C05449=1136.949,196.635,-63.220,-178.213,7.501,148.900
C05450=1136.954,196.386,-63.196,-178.216,7.499,148.901
C05451=1136.958,196.137,-63.172,-178.219,7.496,148.901
C05452=1136.963,195.889,-63.148,-178.222,7.493,148.901
C05453=1136.968,195.639,-63.124,-178.225,7.491,148.901
C05454=1136.973,195.391,-63.100,-178.227,7.488,148.901
C05455=1136.976,195.142,-63.076,-178.230,7.486,148.902
C05456=1136.981,194.893,-63.053,-178.233,7.483,148.902
C05457=1136.986,194.644,-63.028,-178.236,7.481,148.902
C05458=1136.990,194.396,-63.004,-178.239,7.478,148.902
C05459=1136.995,194.147,-62.980,-178.242,7.476,148.902
C05460=1137.000,193.898,-62.956,-178.244,7.474,148.903
C05461=1137.004,193.649,-62.933,-178.247,7.471,148.903
C05462=1137.009,193.401,-62.909,-178.250,7.468,148.903
C05463=1137.013,193.151,-62.885,-178.252,7.466,148.903
C05464=1137.017,192.903,-62.861,-178.256,7.464,148.904
C05465=1137.022,192.654,-62.838,-178.258,7.462,148.904
C05466=1137.026,192.405,-62.814,-178.261,7.459,148.904
C05467=1137.032,192.156,-62.790,-178.264,7.456,148.904
C05468=1137.036,191.908,-62.766,-178.267,7.454,148.905
C05469=1137.041,191.658,-62.742,-178.270,7.452,148.905
C05470=1137.045,191.410,-62.718,-178.273,7.449,148.905
C05471=1137.050,191.161,-62.695,-178.275,7.447,148.905
C05472=1137.055,190.912,-62.671,-178.278,7.444,148.905
C05473=1137.059,190.664,-62.647,-178.281,7.442,148.906
C05474=1137.064,190.415,-62.624,-178.284,7.440,148.906
C05475=1137.068,190.166,-62.600,-178.287,7.437,148.906
C05476=1137.073,189.917,-62.577,-178.290,7.434,148.906
C05477=1137.078,189.668,-62.553,-178.292,7.432,148.907
C05478=1137.082,189.420,-62.529,-178.295,7.429,148.907
C05479=1137.087,189.171,-62.506,-178.298,7.428,148.907
C05480=1137.091,188.922,-62.482,-178.301,7.425,148.907
C05481=1137.096,188.673,-62.459,-178.304,7.422,148.907
C05482=1137.101,188.424,-62.435,-178.306,7.420,148.908
C05483=1137.105,188.175,-62.412,-178.309,7.418,148.908
C05484=1137.110,187.926,-62.388,-178.312,7.416,148.908
C05485=1137.115,187.677,-62.365,-178.315,7.413,148.908
C05486=1137.119,187.429,-62.341,-178.318,7.410,148.909
C05487=1137.124,187.180,-62.318,-178.320,7.408,148.909
C05488=1137.128,186.931,-62.294,-178.323,7.405,148.909
C05489=1137.133,186.682,-62.271,-178.327,7.403,148.909
C05490=1137.137,186.433,-62.247,-178.329,7.401,148.909
C05491=1137.141,186.184,-62.224,-178.332,7.398,148.910
C05492=1137.146,185.935,-62.201,-178.334,7.396,148.910
C05493=1137.151,185.686,-62.177,-178.338,7.394,148.910
C05494=1137.156,185.437,-62.154,-178.341,7.391,148.911
C05495=1137.160,185.188,-62.131,-178.343,7.389,148.911
C05496=1137.165,184.939,-62.107,-178.346,7.387,148.911
C05497=1137.169,184.691,-62.084,-178.349,7.384,148.911
C05498=1137.173,184.442,-62.060,-178.352,7.382,148.912
C05499=1137.178,184.193,-62.037,-178.354,7.380,148.912
C05500=1137.183,183.944,-62.014,-178.357,7.377,148.912
C05501=1137.188,183.674,-61.989,-178.360,7.374,148.912
C05502=1137.193,183.405,-61.964,-178.363,7.372,148.913
C05503=1137.198,183.135,-61.939,-178.367,7.369,148.913
C05504=1137.203,182.866,-61.913,-178.370,7.366,148.913
C05505=1137.208,182.617,-61.890,-178.372,7.365,148.913
C05506=1137.212,182.368,-61.867,-178.375,7.362,148.914
C05507=1137.216,182.119,-61.844,-178.378,7.360,148.914
C05508=1137.221,181.869,-61.821,-178.381,7.358,148.914
C05509=1137.226,181.620,-61.798,-178.383,7.356,148.914
C05510=1137.231,181.372,-61.775,-178.387,7.353,148.915
C05511=1137.235,181.123,-61.752,-178.389,7.351,148.915
C05512=1137.240,180.874,-61.729,-178.392,7.348,148.915
C05513=1137.245,180.625,-61.705,-178.395,7.345,148.915
C05514=1137.249,180.377,-61.683,-178.398,7.344,148.916
C05515=1137.253,180.128,-61.659,-178.401,7.341,148.916
C05516=1137.259,179.879,-61.636,-178.403,7.339,148.916
C05517=1137.263,179.630,-61.614,-178.406,7.337,148.917
C05518=1137.268,179.381,-61.591,-178.409,7.335,148.917
C05519=1137.272,179.132,-61.568,-178.412,7.332,148.917
C05520=1137.276,178.883,-61.545,-178.414,7.330,148.917
C05521=1137.281,178.634,-61.521,-178.418,7.327,148.918
C05522=1137.286,178.385,-61.500,-178.421,7.325,148.918
C05523=1137.291,178.136,-61.476,-178.423,7.323,148.918
C05524=1137.295,177.887,-61.453,-178.426,7.320,148.918
C05525=1137.299,177.639,-61.430,-178.429,7.318,148.918
C05526=1137.305,177.390,-61.408,-178.432,7.316,148.919
C05527=1137.309,177.141,-61.385,-178.435,7.314,148.919
C05528=1137.313,176.892,-61.362,-178.437,7.311,148.919
C05529=1137.318,176.643,-61.338,-178.440,7.309,148.920
C05530=1137.323,176.394,-61.317,-178.443,7.306,148.920
C05531=1137.328,176.145,-61.293,-178.446,7.305,148.920
C05532=1137.332,175.897,-61.271,-178.449,7.302,148.921
C05533=1137.337,175.647,-61.248,-178.451,7.300,148.921
C05534=1137.341,175.399,-61.226,-178.454,7.298,148.921
C05535=1137.346,175.149,-61.203,-178.457,7.295,148.921
C05536=1137.350,174.900,-61.180,-178.460,7.293,148.922
C05537=1137.355,174.651,-61.157,-178.463,7.291,148.922
C05538=1137.360,174.403,-61.135,-178.465,7.288,148.922
C05539=1137.365,174.154,-61.112,-178.468,7.287,148.922
C05540=1137.369,173.904,-61.090,-178.471,7.284,148.923
C05541=1137.374,173.656,-61.067,-178.474,7.282,148.923
C05542=1137.378,173.407,-61.045,-178.477,7.279,148.923
C05543=1137.383,173.158,-61.021,-178.479,7.277,148.923
C05544=1137.388,172.909,-61.000,-178.483,7.275,148.924
C05545=1137.393,172.660,-60.976,-178.485,7.273,148.924
C05546=1137.397,172.411,-60.954,-178.488,7.270,148.924
C05547=1137.401,172.163,-60.932,-178.491,7.269,148.925
C05548=1137.406,171.913,-60.909,-178.494,7.266,148.925
C05549=1137.410,171.664,-60.886,-178.496,7.264,148.925
C05550=1137.416,171.415,-60.864,-178.500,7.261,148.925
C05551=1137.420,171.167,-60.841,-178.502,7.260,148.926
C05552=1137.425,170.918,-60.820,-178.505,7.257,148.926
C05553=1137.430,170.668,-60.797,-178.508,7.255,148.926
C05554=1137.434,170.420,-60.774,-178.511,7.253,148.927
C05555=1137.439,170.171,-60.753,-178.513,7.251,148.927
C05556=1137.444,169.921,-60.730,-178.517,7.248,148.927
C05557=1137.448,169.673,-60.707,-178.519,7.246,148.928
C05558=1137.453,169.424,-60.686,-178.522,7.244,148.928
C05559=1137.458,169.174,-60.663,-178.525,7.242,148.928
C05560=1137.462,168.926,-60.641,-178.528,7.240,148.928
C05561=1137.466,168.677,-60.618,-178.530,7.237,148.929
C05562=1137.472,168.428,-60.596,-178.533,7.235,148.929
C05563=1137.476,168.179,-60.573,-178.536,7.233,148.929
C05564=1137.480,167.930,-60.551,-178.539,7.231,148.929
C05565=1137.486,167.681,-60.529,-178.542,7.228,148.930
C05566=1137.490,167.432,-60.507,-178.545,7.227,148.930
C05567=1137.495,167.183,-60.485,-178.547,7.224,148.930
C05568=1137.499,166.934,-60.463,-178.550,7.222,148.931
C05569=1137.505,166.685,-60.440,-178.553,7.220,148.931
C05570=1137.509,166.436,-60.418,-178.556,7.217,148.931
C05571=1137.514,166.187,-60.397,-178.558,7.216,148.932
C05572=1137.518,165.938,-60.375,-178.562,7.213,148.932
C05573=1137.524,165.689,-60.352,-178.564,7.211,148.932
C05574=1137.527,165.440,-60.330,-178.567,7.208,148.932
C05575=1137.532,165.192,-60.308,-178.570,7.207,148.933
C05576=1137.537,164.942,-60.286,-178.573,7.205,148.933
C05577=1137.542,164.694,-60.264,-178.576,7.202,148.933
C05578=1137.546,164.444,-60.242,-178.578,7.200,148.934
C05579=1137.551,164.195,-60.220,-178.582,7.198,148.934
C05580=1137.556,163.946,-60.198,-178.584,7.196,148.934
C05581=1137.561,163.697,-60.176,-178.587,7.193,148.935
C05582=1137.565,163.448,-60.154,-178.590,7.192,148.935
C05583=1137.570,163.199,-60.132,-178.592,7.190,148.935
C05584=1137.574,162.950,-60.110,-178.595,7.187,148.935
C05585=1137.579,162.702,-60.089,-178.598,7.185,148.936
C05586=1137.583,162.452,-60.067,-178.601,7.183,148.936
C05587=1137.588,162.204,-60.045,-178.604,7.181,148.936
C05588=1137.592,161.954,-60.023,-178.606,7.179,148.937
C05589=1137.598,161.705,-60.001,-178.610,7.176,148.937
C05590=1137.602,161.456,-59.978,-178.612,7.175,148.937
C05591=1137.607,161.207,-59.957,-178.615,7.172,148.938
C05592=1137.612,160.959,-59.935,-178.618,7.170,148.938
C05593=1137.616,160.709,-59.913,-178.620,7.168,148.938
C05594=1137.621,160.461,-59.891,-178.624,7.166,148.939
C05595=1137.625,160.211,-59.869,-178.626,7.164,148.939
C05596=1137.630,159.962,-59.848,-178.629,7.161,148.939
C05597=1137.635,159.713,-59.827,-178.632,7.160,148.940
C05598=1137.640,159.464,-59.805,-178.635,7.158,148.940
C05599=1137.644,159.215,-59.783,-178.638,7.155,148.940
C05600=1137.649,158.966,-59.761,-178.640,7.153,148.941
C05601=1137.654,158.717,-59.739,-178.644,7.151,148.941
C05602=1137.659,158.468,-59.718,-178.646,7.149,148.941
C05603=1137.663,158.219,-59.696,-178.649,7.147,148.941
C05604=1137.668,157.970,-59.675,-178.652,7.145,148.942
C05605=1137.673,157.701,-59.652,-178.655,7.143,148.942
C05606=1137.678,157.432,-59.628,-178.658,7.140,148.943
C05607=1137.683,157.163,-59.605,-178.661,7.138,148.943
C05608=1137.688,156.894,-59.582,-178.664,7.136,148.943
C05609=1137.693,156.645,-59.560,-178.667,7.134,148.944
C05610=1137.698,156.397,-59.538,-178.669,7.131,148.944
C05611=1137.702,156.147,-59.517,-178.672,7.130,148.944
C05612=1137.706,155.898,-59.496,-178.675,7.127,148.945
C05613=1137.711,155.650,-59.474,-178.678,7.126,148.945
C05614=1137.716,155.400,-59.453,-178.680,7.123,148.945
C05615=1137.721,155.151,-59.431,-178.684,7.121,148.945
C05616=1137.726,154.903,-59.409,-178.686,7.119,148.946
C05617=1137.730,154.653,-59.388,-178.689,7.118,148.946
C05618=1137.735,154.404,-59.366,-178.692,7.115,148.947
C05619=1137.740,154.155,-59.346,-178.695,7.113,148.947
C05620=1137.744,153.906,-59.324,-178.697,7.111,148.947
C05621=1137.749,153.656,-59.303,-178.701,7.109,148.947
C05622=1137.754,153.408,-59.281,-178.703,7.107,148.948
C05623=1137.759,153.159,-59.260,-178.706,7.105,148.948
C05624=1137.763,152.910,-59.239,-178.709,7.102,148.948
C05625=1137.767,152.661,-59.217,-178.712,7.101,148.949
C05626=1137.773,152.412,-59.196,-178.714,7.099,148.949
C05627=1137.777,152.163,-59.175,-178.718,7.096,148.950
C05628=1137.783,151.914,-59.154,-178.720,7.095,148.950
C05629=1137.786,151.665,-59.132,-178.723,7.093,148.950
C05630=1137.791,151.415,-59.111,-178.726,7.090,148.950
C05631=1137.796,151.166,-59.090,-178.729,7.088,148.951
C05632=1137.801,150.918,-59.069,-178.731,7.087,148.951
C05633=1137.806,150.669,-59.048,-178.735,7.084,148.952
C05634=1137.810,150.419,-59.026,-178.737,7.082,148.952
C05635=1137.815,150.170,-59.005,-178.740,7.080,148.952
C05636=1137.820,149.921,-58.985,-178.743,7.078,148.953
C05637=1137.825,149.672,-58.963,-178.746,7.076,148.953
C05638=1137.830,149.423,-58.942,-178.748,7.075,148.953
C05639=1137.834,149.173,-58.921,-178.751,7.073,148.954
C05640=1137.838,148.925,-58.900,-178.754,7.070,148.954
C05641=1137.844,148.676,-58.879,-178.757,7.068,148.954
C05642=1137.848,148.427,-58.858,-178.759,7.067,148.955
C05643=1137.853,148.178,-58.837,-178.763,7.064,148.955
C05644=1137.858,147.929,-58.816,-178.765,7.062,148.955
C05645=1137.862,147.679,-58.795,-178.768,7.061,148.956
C05646=1137.867,147.430,-58.773,-178.770,7.059,148.956
C05647=1137.871,147.181,-58.753,-178.774,7.056,148.956
C05648=1137.876,146.932,-58.732,-178.776,7.054,148.957
C05649=1137.882,146.683,-58.711,-178.779,7.053,148.957
C05650=1137.886,146.434,-58.691,-178.782,7.050,148.957
C05651=1137.891,146.185,-58.669,-178.785,7.048,148.958
C05652=1137.895,145.936,-58.649,-178.788,7.047,148.958
C05653=1137.900,145.687,-58.628,-178.790,7.045,148.958
C05654=1137.904,145.437,-58.607,-178.793,7.042,148.959
C05655=1137.910,145.188,-58.586,-178.796,7.040,148.959
C05656=1137.914,144.940,-58.564,-178.799,7.039,148.959
C05657=1137.919,144.691,-58.544,-178.802,7.036,148.960
C05658=1137.924,144.441,-58.523,-178.805,7.035,148.960
C05659=1137.928,144.192,-58.503,-178.807,7.033,148.961
C05660=1137.934,143.943,-58.482,-178.810,7.031,148.961
C05661=1137.938,143.694,-58.461,-178.813,7.028,148.961
C05662=1137.943,143.445,-58.440,-178.816,7.027,148.962
C05663=1137.948,143.196,-58.420,-178.818,7.025,148.962
C05664=1137.952,142.947,-58.399,-178.821,7.023,148.962
C05665=1137.957,142.698,-58.378,-178.824,7.021,148.963
C05666=1137.962,142.449,-58.358,-178.827,7.019,148.963
C05667=1137.967,142.200,-58.337,-178.830,7.017,148.963
C05668=1137.971,141.951,-58.317,-178.832,7.015,148.964
C05669=1137.976,141.701,-58.296,-178.835,7.013,148.964
C05670=1137.980,141.452,-58.275,-178.838,7.011,148.964
C05671=1137.985,141.203,-58.255,-178.841,7.009,148.965
C05672=1137.990,140.953,-58.234,-178.844,7.008,148.965
C05673=1137.994,140.705,-58.213,-178.846,7.006,148.966
C05674=1138.000,140.455,-58.192,-178.850,7.003,148.966
C05675=1138.004,140.206,-58.172,-178.852,7.002,148.966
C05676=1138.008,139.957,-58.152,-178.855,7.000,148.967
C05677=1138.014,139.708,-58.131,-178.857,6.998,148.967
C05678=1138.019,139.460,-58.111,-178.861,6.995,148.967
C05679=1138.023,139.211,-58.090,-178.863,6.994,148.968
C05680=1138.028,138.962,-58.069,-178.866,6.992,148.968
C05681=1138.033,138.712,-58.050,-178.869,6.990,148.968
C05682=1138.037,138.463,-58.029,-178.871,6.989,148.969
C05683=1138.043,138.214,-58.008,-178.875,6.986,148.969
C05684=1138.047,137.965,-57.988,-178.878,6.984,148.970
C05685=1138.051,137.716,-57.968,-178.880,6.983,148.970
C05686=1138.057,137.466,-57.947,-178.883,6.981,148.970
C05687=1138.061,137.217,-57.927,-178.886,6.978,148.971
C05688=1138.066,136.968,-57.907,-178.889,6.976,148.971
C05689=1138.070,136.719,-57.886,-178.891,6.975,148.971
C05690=1138.075,136.470,-57.865,-178.894,6.973,148.972
C05691=1138.080,136.220,-57.846,-178.897,6.971,148.972
C05692=1138.085,135.972,-57.825,-178.900,6.969,148.973
C05693=1138.089,135.723,-57.805,-178.903,6.967,148.973
C05694=1138.095,135.473,-57.785,-178.905,6.965,148.973
C05695=1138.100,135.224,-57.765,-178.908,6.964,148.974
C05696=1138.104,134.975,-57.744,-178.911,6.962,148.974
C05697=1138.109,134.726,-57.725,-178.914,6.960,148.975
C05698=1138.114,134.477,-57.704,-178.917,6.958,148.975
C05699=1138.118,134.228,-57.683,-178.920,6.956,148.975
C05700=1138.123,133.978,-57.664,-178.922,6.954,148.976
C05701=1138.128,133.729,-57.643,-178.925,6.953,148.976
C05702=1138.133,133.481,-57.623,-178.928,6.951,148.976
C05703=1138.137,133.231,-57.604,-178.931,6.948,148.977
C05704=1138.142,132.982,-57.583,-178.933,6.946,148.977
C05705=1138.147,132.733,-57.563,-178.936,6.945,148.977
C05706=1138.152,132.484,-57.543,-178.939,6.943,148.978
C05707=1138.156,132.234,-57.523,-178.942,6.941,148.978
C05708=1138.161,131.986,-57.503,-178.944,6.940,148.979
C05709=1138.167,131.717,-57.481,-178.948,6.937,148.979
C05710=1138.172,131.449,-57.459,-178.950,6.936,148.979
C05711=1138.177,131.180,-57.438,-178.954,6.933,148.980
C05712=1138.182,130.911,-57.417,-178.957,6.932,148.980
C05713=1138.187,130.662,-57.396,-178.960,6.930,148.981
C05714=1138.191,130.413,-57.377,-178.962,6.928,148.981
C05715=1138.196,130.164,-57.356,-178.965,6.927,148.982
C05716=1138.201,129.915,-57.337,-178.968,6.924,148.982
C05717=1138.206,129.666,-57.317,-178.971,6.922,148.982
C05718=1138.210,129.416,-57.297,-178.973,6.920,148.983
C05719=1138.215,129.167,-57.277,-178.976,6.919,148.983
C05720=1138.220,128.919,-57.257,-178.979,6.917,148.983
C05721=1138.225,128.669,-57.238,-178.981,6.915,148.984
C05722=1138.229,128.420,-57.217,-178.984,6.914,148.984
C05723=1138.234,128.170,-57.198,-178.987,6.911,148.985
C05724=1138.239,127.922,-57.178,-178.990,6.909,148.985
C05725=1138.244,127.673,-57.158,-178.993,6.908,148.985
C05726=1138.249,127.423,-57.138,-178.996,6.906,148.986
C05727=1138.253,127.173,-57.119,-178.998,6.904,148.986
C05728=1138.258,126.925,-57.099,-179.001,6.903,148.986
C05729=1138.263,126.676,-57.079,-179.004,6.901,148.987
C05730=1138.268,126.426,-57.059,-179.007,6.899,148.987
C05731=1138.273,126.177,-57.040,-179.010,6.897,148.988
C05732=1138.278,125.928,-57.020,-179.013,6.895,148.988
C05733=1138.282,125.679,-57.000,-179.015,6.893,148.988
C05734=1138.287,125.429,-56.980,-179.018,6.892,148.989
C05735=1138.293,125.180,-56.961,-179.021,6.890,148.989
C05736=1138.297,124.931,-56.941,-179.023,6.888,148.990
C05737=1138.302,124.682,-56.921,-179.026,6.887,148.990
C05738=1138.306,124.433,-56.902,-179.029,6.885,148.990
C05739=1138.311,124.184,-56.883,-179.032,6.883,148.991
C05740=1138.316,123.934,-56.863,-179.035,6.881,148.991
C05741=1138.321,123.686,-56.843,-179.038,6.879,148.992
C05742=1138.326,123.436,-56.823,-179.040,6.877,148.992
C05743=1138.330,123.187,-56.804,-179.043,6.876,148.992
C05744=1138.336,122.938,-56.784,-179.046,6.874,148.993
C05745=1138.340,122.689,-56.765,-179.049,6.872,148.993
C05746=1138.344,122.439,-56.746,-179.051,6.871,148.994
C05747=1138.350,122.190,-56.726,-179.054,6.869,148.994
C05748=1138.355,121.941,-56.707,-179.057,6.867,148.994
C05749=1138.359,121.691,-56.687,-179.059,6.866,148.995
C05750=1138.364,121.442,-56.668,-179.062,6.864,148.995
C05751=1138.369,121.193,-56.649,-179.066,6.861,148.996
C05752=1138.374,120.945,-56.629,-179.068,6.860,148.996
C05753=1138.378,120.695,-56.609,-179.071,6.858,148.996
C05754=1138.383,120.445,-56.589,-179.074,6.856,148.997
C05755=1138.388,120.197,-56.571,-179.076,6.855,148.997
C05756=1138.392,119.947,-56.551,-179.079,6.853,148.998
C05757=1138.398,119.698,-56.532,-179.082,6.851,148.998
C05758=1138.403,119.448,-56.513,-179.085,6.850,148.998
C05759=1138.407,119.200,-56.494,-179.088,6.848,148.999
C05760=1138.412,118.950,-56.474,-179.091,6.847,149.000
C05761=1138.417,118.701,-56.455,-179.093,6.845,149.000
C05762=1138.422,118.452,-56.436,-179.096,6.843,149.000
C05763=1138.426,118.202,-56.416,-179.099,6.841,149.001
C05764=1138.432,117.954,-56.397,-179.101,6.840,149.001
C05765=1138.436,117.704,-56.378,-179.104,6.838,149.002
C05766=1138.441,117.455,-56.359,-179.107,6.836,149.002
C05767=1138.446,117.206,-56.339,-179.110,6.834,149.002
C05768=1138.450,116.957,-56.320,-179.113,6.832,149.003
C05769=1138.455,116.707,-56.302,-179.116,6.831,149.003
C05770=1138.461,116.458,-56.282,-179.118,6.829,149.004
C05771=1138.465,116.209,-56.263,-179.121,6.827,149.004
C05772=1138.470,115.960,-56.244,-179.124,6.825,149.004
C05773=1138.475,115.711,-56.224,-179.127,6.824,149.005
C05774=1138.480,115.461,-56.206,-179.129,6.822,149.005
C05775=1138.484,115.212,-56.187,-179.132,6.820,149.006
C05776=1138.489,114.963,-56.168,-179.135,6.819,149.006
C05777=1138.494,114.714,-56.148,-179.138,6.817,149.006
C05778=1138.499,114.464,-56.130,-179.140,6.815,149.007
C05779=1138.503,114.215,-56.111,-179.143,6.814,149.007
C05780=1138.509,113.966,-56.091,-179.146,6.812,149.008
C05781=1138.513,113.717,-56.072,-179.149,6.811,149.008
C05782=1138.518,113.467,-56.054,-179.152,6.809,149.009
C05783=1138.523,113.219,-56.035,-179.154,6.807,149.009
C05784=1138.528,112.969,-56.015,-179.157,6.806,149.009
C05785=1138.533,112.720,-55.997,-179.160,6.804,149.010
C05786=1138.538,112.471,-55.978,-179.163,6.802,149.010
C05787=1138.543,112.222,-55.958,-179.165,6.801,149.011
C05788=1138.547,111.972,-55.940,-179.168,6.799,149.011
C05789=1138.552,111.723,-55.921,-179.171,6.797,149.012
C05790=1138.557,111.474,-55.903,-179.173,6.796,149.012
C05791=1138.562,111.224,-55.883,-179.176,6.794,149.012
C05792=1138.567,110.976,-55.864,-179.179,6.792,149.013
C05793=1138.572,110.725,-55.845,-179.182,6.791,149.013
C05794=1138.576,110.477,-55.827,-179.185,6.789,149.014
C05795=1138.582,110.227,-55.808,-179.188,6.787,149.014
C05796=1138.586,109.978,-55.789,-179.190,6.786,149.015
C05797=1138.591,109.729,-55.771,-179.193,6.784,149.015
C05798=1138.596,109.479,-55.752,-179.196,6.782,149.015
C05799=1138.601,109.230,-55.734,-179.199,6.781,149.016
C05800=1138.606,108.981,-55.714,-179.201,6.779,149.016
C05801=1138.610,108.731,-55.696,-179.204,6.777,149.017
C05802=1138.615,108.483,-55.677,-179.207,6.776,149.017
C05803=1138.621,108.233,-55.659,-179.209,6.774,149.017
C05804=1138.625,107.984,-55.640,-179.212,6.772,149.018
C05805=1138.630,107.735,-55.621,-179.215,6.771,149.019
C05806=1138.635,107.486,-55.602,-179.218,6.769,149.019
C05807=1138.639,107.236,-55.584,-179.221,6.768,149.019
C05808=1138.644,106.987,-55.565,-179.224,6.766,149.020
C05809=1138.649,106.738,-55.547,-179.226,6.764,149.020
C05810=1138.654,106.488,-55.528,-179.229,6.763,149.021
C05811=1138.659,106.239,-55.509,-179.232,6.761,149.021
C05812=1138.664,105.990,-55.491,-179.235,6.759,149.021
C05813=1138.668,105.721,-55.471,-179.238,6.758,149.022
C05814=1138.674,105.453,-55.451,-179.240,6.756,149.022
C05815=1138.679,105.185,-55.431,-179.243,6.755,149.023
C05816=1138.685,104.917,-55.411,-179.246,6.753,149.023
C05817=1138.690,104.667,-55.393,-179.249,6.752,149.024
C05818=1138.694,104.418,-55.374,-179.252,6.750,149.024
C05819=1138.699,104.169,-55.356,-179.255,6.748,149.025
C05820=1138.704,103.919,-55.338,-179.257,6.747,149.025
C05821=1138.708,103.670,-55.318,-179.260,6.745,149.026
C05822=1138.713,103.421,-55.301,-179.263,6.743,149.026
C05823=1138.719,103.172,-55.282,-179.266,6.742,149.026
C05824=1138.724,102.922,-55.264,-179.268,6.740,149.027
C05825=1138.728,102.673,-55.245,-179.271,6.738,149.027
C05826=1138.733,102.424,-55.227,-179.274,6.737,149.028
C05827=1138.738,102.174,-55.208,-179.277,6.735,149.028
C05828=1138.743,101.925,-55.190,-179.280,6.734,149.029
C05829=1138.748,101.676,-55.172,-179.282,6.732,149.029
C05830=1138.753,101.426,-55.154,-179.285,6.730,149.029
C05831=1138.757,101.178,-55.135,-179.287,6.729,149.030
C05832=1138.763,100.928,-55.117,-179.290,6.728,149.030
C05833=1138.768,100.679,-55.099,-179.293,6.726,149.031
C05834=1138.773,100.430,-55.081,-179.296,6.725,149.031
C05835=1138.777,100.180,-55.062,-179.299,6.723,149.032
C05836=1138.782,99.931,-55.044,-179.302,6.721,149.032
C05837=1138.787,99.682,-55.026,-179.304,6.720,149.033
C05838=1138.792,99.432,-55.009,-179.307,6.718,149.033
C05839=1138.797,99.184,-54.989,-179.310,6.716,149.033
C05840=1138.801,98.934,-54.971,-179.313,6.715,149.034
C05841=1138.806,98.684,-54.953,-179.316,6.713,149.035
C05842=1138.811,98.435,-54.935,-179.318,6.712,149.035
C05843=1138.816,98.186,-54.917,-179.321,6.711,149.035
C05844=1138.821,97.937,-54.899,-179.323,6.709,149.036
C05845=1138.826,97.688,-54.881,-179.326,6.707,149.036
C05846=1138.831,97.439,-54.863,-179.329,6.706,149.037
C05847=1138.835,97.189,-54.845,-179.332,6.704,149.037
C05848=1138.840,96.940,-54.827,-179.335,6.703,149.038
C05849=1138.845,96.690,-54.809,-179.337,6.701,149.038
C05850=1138.850,96.441,-54.791,-179.340,6.699,149.038
C05851=1138.855,96.192,-54.773,-179.343,6.698,149.039
C05852=1138.860,95.942,-54.755,-179.345,6.697,149.039
C05853=1138.865,95.693,-54.737,-179.348,6.696,149.040
C05854=1138.870,95.444,-54.719,-179.351,6.694,149.040
C05855=1138.875,95.194,-54.701,-179.354,6.692,149.041
C05856=1138.880,94.945,-54.683,-179.356,6.691,149.041
C05857=1138.884,94.696,-54.665,-179.359,6.689,149.042
C05858=1138.889,94.446,-54.647,-179.362,6.687,149.042
C05859=1138.894,94.197,-54.629,-179.365,6.686,149.042
C05860=1138.899,93.948,-54.611,-179.367,6.685,149.043
C05861=1138.904,93.698,-54.594,-179.370,6.683,149.044
C05862=1138.909,93.449,-54.576,-179.373,6.682,149.044
C05863=1138.914,93.200,-54.558,-179.376,6.680,149.044
C05864=1138.919,92.951,-54.540,-179.378,6.678,149.045
C05865=1138.923,92.702,-54.522,-179.381,6.677,149.045
C05866=1138.929,92.452,-54.505,-179.384,6.675,149.046
C05867=1138.934,92.203,-54.487,-179.386,6.675,149.046
C05868=1138.939,91.953,-54.469,-179.389,6.673,149.047
C05869=1138.943,91.704,-54.451,-179.392,6.671,149.047
C05870=1138.949,91.455,-54.434,-179.395,6.670,149.048
C05871=1138.954,91.205,-54.416,-179.398,6.668,149.048
C05872=1138.958,90.956,-54.398,-179.401,6.667,149.049
C05873=1138.963,90.707,-54.380,-179.403,6.666,149.049
C05874=1138.968,90.458,-54.363,-179.405,6.664,149.049
C05875=1138.973,90.208,-54.345,-179.408,6.662,149.050
C05876=1138.978,89.959,-54.327,-179.411,6.661,149.051
C05877=1138.983,89.709,-54.310,-179.414,6.659,149.051
C05878=1138.988,89.460,-54.292,-179.417,6.658,149.051
C05879=1138.992,89.211,-54.274,-179.420,6.656,149.052
C05880=1138.997,88.962,-54.257,-179.422,6.655,149.052
C05881=1139.002,88.712,-54.239,-179.425,6.654,149.053
C05882=1139.007,88.463,-54.222,-179.428,6.652,149.053
C05883=1139.012,88.213,-54.204,-179.430,6.651,149.054
C05884=1139.016,87.965,-54.187,-179.433,6.649,149.054
C05885=1139.022,87.715,-54.169,-179.435,6.648,149.055
C05886=1139.027,87.466,-54.151,-179.438,6.646,149.055
C05887=1139.032,87.216,-54.134,-179.441,6.645,149.056
C05888=1139.037,86.967,-54.116,-179.444,6.643,149.056
C05889=1139.041,86.717,-54.099,-179.447,6.642,149.056
C05890=1139.046,86.468,-54.081,-179.450,6.640,149.057
C05891=1139.051,86.219,-54.063,-179.452,6.639,149.057
C05892=1139.056,85.969,-54.046,-179.455,6.638,149.058
C05893=1139.060,85.720,-54.029,-179.458,6.636,149.058
C05894=1139.066,85.470,-54.012,-179.460,6.635,149.059
C05895=1139.071,85.221,-53.994,-179.463,6.633,149.059
C05896=1139.076,84.972,-53.977,-179.465,6.632,149.060
C05897=1139.081,84.723,-53.960,-179.469,6.631,149.060
C05898=1139.086,84.473,-53.942,-179.471,6.629,149.061
C05899=1139.090,84.224,-53.925,-179.474,6.628,149.061
C05900=1139.095,83.975,-53.907,-179.477,6.626,149.062
C05901=1139.100,83.725,-53.890,-179.479,6.625,149.062
C05902=1139.105,83.476,-53.873,-179.482,6.624,149.063
C05903=1139.110,83.226,-53.855,-179.485,6.622,149.063
C05904=1139.116,82.977,-53.839,-179.488,6.620,149.064
C05905=1139.120,82.728,-53.821,-179.490,6.620,149.064
C05906=1139.125,82.478,-53.804,-179.493,6.618,149.065
C05907=1139.130,82.229,-53.787,-179.496,6.617,149.065
C05908=1139.134,81.980,-53.769,-179.498,6.615,149.065
C05909=1139.140,81.730,-53.752,-179.501,6.613,149.066
C05910=1139.144,81.481,-53.735,-179.503,6.612,149.066
C05911=1139.150,81.232,-53.718,-179.507,6.611,149.067
C05912=1139.155,80.982,-53.700,-179.509,6.609,149.067
C05913=1139.159,80.733,-53.684,-179.512,6.608,149.068
C05914=1139.164,80.484,-53.666,-179.514,6.607,149.068
C05915=1139.169,80.234,-53.649,-179.517,6.606,149.069
C05916=1139.174,79.985,-53.632,-179.520,6.604,149.069
C05917=1139.180,79.716,-53.614,-179.523,6.602,149.070
C05918=1139.185,79.448,-53.595,-179.526,6.601,149.070
C05919=1139.190,79.179,-53.577,-179.529,6.599,149.071
C05920=1139.195,78.911,-53.559,-179.532,6.598,149.071
C05921=1139.200,78.662,-53.541,-179.535,6.596,149.072
C05922=1139.205,78.413,-53.525,-179.537,6.596,149.072
C05923=1139.210,78.163,-53.507,-179.540,6.594,149.073
C05924=1139.216,77.913,-53.490,-179.542,6.592,149.073
C05925=1139.220,77.664,-53.474,-179.546,6.591,149.074
C05926=1139.224,77.415,-53.456,-179.548,6.590,149.074
C05927=1139.230,77.166,-53.439,-179.551,6.588,149.075
C05928=1139.235,76.916,-53.423,-179.553,6.587,149.075
C05929=1139.240,76.667,-53.405,-179.557,6.585,149.076
C05930=1139.245,76.418,-53.389,-179.559,6.585,149.076
C05931=1139.250,76.168,-53.372,-179.561,6.583,149.077
C05932=1139.255,75.919,-53.355,-179.564,6.581,149.077
C05933=1139.260,75.669,-53.338,-179.567,6.581,149.078
C05934=1139.265,75.420,-53.321,-179.570,6.579,149.078
C05935=1139.270,75.170,-53.304,-179.572,6.578,149.079
C05936=1139.274,74.921,-53.287,-179.575,6.576,149.079
C05937=1139.279,74.672,-53.270,-179.578,6.575,149.080
C05938=1139.285,74.423,-53.253,-179.580,6.574,149.080
C05939=1139.289,74.173,-53.237,-179.583,6.572,149.081
C05940=1139.294,73.923,-53.219,-179.586,6.570,149.081
C05941=1139.299,73.675,-53.203,-179.589,6.570,149.082
C05942=1139.304,73.425,-53.186,-179.591,6.568,149.082
C05943=1139.309,73.175,-53.169,-179.594,6.567,149.083
C05944=1139.314,72.927,-53.153,-179.596,6.566,149.083
C05945=1139.319,72.676,-53.137,-179.599,6.564,149.084
C05946=1139.324,72.427,-53.120,-179.602,6.563,149.084
C05947=1139.329,72.178,-53.103,-179.604,6.562,149.084
C05948=1139.334,71.928,-53.087,-179.607,6.560,149.085
C05949=1139.339,71.679,-53.069,-179.610,6.559,149.086
C05950=1139.344,71.430,-53.053,-179.613,6.557,149.086
C05951=1139.348,71.180,-53.036,-179.615,6.557,149.086
C05952=1139.354,70.931,-53.019,-179.618,6.555,149.087
C05953=1139.359,70.682,-53.003,-179.621,6.554,149.088
C05954=1139.363,70.432,-52.986,-179.623,6.553,149.088
C05955=1139.369,70.182,-52.970,-179.626,6.551,149.088
C05956=1139.374,69.933,-52.953,-179.629,6.550,149.089
C05957=1139.378,69.684,-52.937,-179.632,6.549,149.089
C05958=1139.383,69.435,-52.920,-179.634,6.547,149.090
C05959=1139.389,69.185,-52.903,-179.637,6.546,149.090
C05960=1139.393,68.936,-52.886,-179.640,6.545,149.091
C05961=1139.398,68.686,-52.871,-179.642,6.544,149.091
C05962=1139.403,68.437,-52.854,-179.645,6.542,149.092
C05963=1139.409,68.188,-52.837,-179.647,6.541,149.092
C05964=1139.413,67.938,-52.821,-179.651,6.540,149.093
C05965=1139.418,67.688,-52.805,-179.653,6.538,149.093
C05966=1139.423,67.439,-52.788,-179.656,6.536,149.094
C05967=1139.428,67.190,-52.772,-179.658,6.536,149.094
C05968=1139.433,66.941,-52.755,-179.661,6.534,149.095
C05969=1139.438,66.691,-52.739,-179.664,6.533,149.095
C05970=1139.443,66.442,-52.722,-179.666,6.532,149.096
C05971=1139.448,66.192,-52.706,-179.670,6.531,149.096
C05972=1139.453,65.943,-52.690,-179.672,6.530,149.097
C05973=1139.458,65.693,-52.674,-179.674,6.528,149.097
C05974=1139.463,65.444,-52.656,-179.677,6.526,149.098
C05975=1139.468,65.194,-52.641,-179.680,6.526,149.098
C05976=1139.473,64.945,-52.624,-179.683,6.524,149.099
C05977=1139.478,64.696,-52.608,-179.685,6.523,149.099
C05978=1139.483,64.446,-52.592,-179.688,6.522,149.100
C05979=1139.488,64.197,-52.575,-179.691,6.520,149.100
C05980=1139.492,63.948,-52.559,-179.693,6.519,149.101
C05981=1139.498,63.698,-52.543,-179.696,6.518,149.101
C05982=1139.502,63.449,-52.527,-179.699,6.517,149.102
C05983=1139.508,63.199,-52.510,-179.702,6.515,149.102
C05984=1139.513,62.949,-52.494,-179.704,6.514,149.103
C05985=1139.518,62.700,-52.478,-179.707,6.513,149.103
C05986=1139.522,62.451,-52.461,-179.709,6.512,149.104
C05987=1139.528,62.202,-52.445,-179.712,6.510,149.104
C05988=1139.532,61.952,-52.429,-179.715,6.509,149.105
C05989=1139.537,61.703,-52.413,-179.717,6.508,149.105
C05990=1139.542,61.453,-52.397,-179.720,6.507,149.106
C05991=1139.547,61.204,-52.381,-179.723,6.505,149.106
C05992=1139.553,60.955,-52.365,-179.725,6.505,149.107
C05993=1139.557,60.705,-52.348,-179.728,6.503,149.107
C05994=1139.563,60.456,-52.333,-179.730,6.502,149.108
C05995=1139.567,60.206,-52.317,-179.734,6.501,149.109
C05996=1139.572,59.957,-52.301,-179.736,6.499,149.109
C05997=1139.577,59.707,-52.285,-179.738,6.498,149.109
C05998=1139.582,59.458,-52.268,-179.741,6.497,149.110
C05999=1139.587,59.208,-52.252,-179.744,6.495,149.111
C06000=1139.592,58.959,-52.236,-179.747,6.495,149.111
C06001=1139.598,58.710,-52.220,-179.749,6.493,149.111
C06002=1139.602,58.460,-52.204,-179.752,6.492,149.112
C06003=1139.607,58.211,-52.188,-179.755,6.491,149.112
C06004=1139.612,57.961,-52.172,-179.758,6.489,149.113
C06005=1139.618,57.711,-52.157,-179.760,6.489,149.114
C06006=1139.623,57.463,-52.140,-179.763,6.487,149.114
C06007=1139.627,57.212,-52.124,-179.765,6.486,149.114
C06008=1139.633,56.963,-52.109,-179.768,6.485,149.115
C06009=1139.637,56.714,-52.093,-179.771,6.483,149.116
C06010=1139.642,56.464,-52.077,-179.773,6.482,149.116
C06011=1139.647,56.215,-52.062,-179.776,6.481,149.116
C06012=1139.652,55.966,-52.045,-179.779,6.480,149.117
C06013=1139.657,55.716,-52.029,-179.781,6.479,149.118
C06014=1139.663,55.467,-52.014,-179.784,6.478,149.118
C06015=1139.667,55.217,-51.998,-179.787,6.477,149.119
C06016=1139.672,54.968,-51.981,-179.790,6.475,149.119
C06017=1139.678,54.718,-51.966,-179.792,6.474,149.120
C06018=1139.682,54.469,-51.950,-179.795,6.473,149.120
C06019=1139.687,54.219,-51.935,-179.797,6.472,149.121
C06020=1139.692,53.970,-51.919,-179.800,6.470,149.121
C06021=1139.698,53.701,-51.902,-179.803,6.469,149.122
C06022=1139.703,53.432,-51.885,-179.805,6.468,149.122
C06023=1139.709,53.164,-51.868,-179.808,6.467,149.123
C06024=1139.714,52.895,-51.851,-179.811,6.465,149.123
C06025=1139.719,52.646,-51.836,-179.814,6.464,149.124
C06026=1139.724,52.396,-51.820,-179.817,6.463,149.124
C06027=1139.729,52.147,-51.804,-179.819,6.462,149.125
C06028=1139.734,51.898,-51.788,-179.822,6.461,149.126
C06029=1139.740,51.648,-51.772,-179.825,6.459,149.126
C06030=1139.744,51.399,-51.757,-179.827,6.459,149.126
C06031=1139.749,51.149,-51.741,-179.830,6.457,149.127
C06032=1139.754,50.900,-51.726,-179.832,6.457,149.128
C06033=1139.759,50.650,-51.710,-179.835,6.455,149.128
C06034=1139.764,50.401,-51.695,-179.837,6.454,149.128
C06035=1139.769,50.151,-51.679,-179.840,6.453,149.129
C06036=1139.775,49.902,-51.664,-179.843,6.451,149.130
C06037=1139.779,49.652,-51.648,-179.845,6.450,149.130
C06038=1139.784,49.403,-51.633,-179.849,6.449,149.131
C06039=1139.789,49.153,-51.617,-179.851,6.448,149.131
C06040=1139.794,48.904,-51.602,-179.854,6.447,149.132
C06041=1139.799,48.654,-51.586,-179.856,6.446,149.132
C06042=1139.804,48.405,-51.571,-179.859,6.444,149.133
C06043=1139.810,48.155,-51.555,-179.861,6.444,149.133
C06044=1139.814,47.906,-51.540,-179.864,6.442,149.134
C06045=1139.820,47.657,-51.525,-179.866,6.442,149.134
C06046=1139.824,47.407,-51.509,-179.869,6.440,149.135
C06047=1139.829,47.158,-51.494,-179.872,6.439,149.135
C06048=1139.834,46.908,-51.478,-179.875,6.438,149.136
C06049=1139.839,46.659,-51.463,-179.877,6.437,149.136
C06050=1139.845,46.410,-51.447,-179.880,6.436,149.137
C06051=1139.849,46.160,-51.431,-179.882,6.435,149.137
C06052=1139.854,45.910,-51.416,-179.885,6.433,149.138
C06053=1139.859,45.661,-51.401,-179.888,6.432,149.138
C06054=1139.864,45.412,-51.386,-179.890,6.431,149.139
C06055=1139.870,45.162,-51.371,-179.893,6.429,149.139
C06056=1139.874,44.912,-51.355,-179.896,6.429,149.140
C06057=1139.879,44.663,-51.340,-179.899,6.427,149.140
C06058=1139.885,44.413,-51.324,-179.901,6.427,149.141
C06059=1139.889,44.164,-51.309,-179.904,6.425,149.142
C06060=1139.895,43.915,-51.294,-179.906,6.424,149.142
C06061=1139.900,43.665,-51.279,-179.909,6.423,149.143
C06062=1139.905,43.416,-51.264,-179.911,6.422,149.143
C06063=1139.910,43.166,-51.248,-179.914,6.421,149.144
C06064=1139.914,42.917,-51.233,-179.917,6.420,149.144
C06065=1139.920,42.667,-51.218,-179.920,6.419,149.145
C06066=1139.925,42.417,-51.203,-179.922,6.418,149.145
C06067=1139.930,42.168,-51.188,-179.924,6.417,149.146
C06068=1139.935,41.919,-51.173,-179.927,6.416,149.146
C06069=1139.940,41.670,-51.157,-179.929,6.415,149.147
C06070=1139.945,41.420,-51.143,-179.933,6.414,149.147
C06071=1139.950,41.170,-51.127,-179.935,6.413,149.148
C06072=1139.954,40.921,-51.112,-179.938,6.411,149.148
C06073=1139.960,40.671,-51.097,-179.940,6.411,149.149
C06074=1139.965,40.422,-51.082,-179.943,6.409,149.149
C06075=1139.970,40.172,-51.066,-179.945,6.408,149.150
C06076=1139.975,39.922,-51.052,-179.948,6.407,149.151
C06077=1139.981,39.673,-51.037,-179.951,6.406,149.151
C06078=1139.985,39.424,-51.022,-179.953,6.404,149.151
C06079=1139.990,39.174,-51.007,-179.956,6.404,149.152
C06080=1139.996,38.925,-50.992,-179.959,6.402,149.153
C06081=1140.000,38.676,-50.977,-179.961,6.402,149.153
C06082=1140.006,38.426,-50.962,-179.964,6.400,149.154
C06083=1140.011,38.177,-50.947,-179.966,6.399,149.154
C06084=1140.016,37.927,-50.932,-179.969,6.399,149.155
C06085=1140.021,37.677,-50.917,-179.972,6.397,149.155
C06086=1140.026,37.428,-50.903,-179.974,6.397,149.156
C06087=1140.031,37.178,-50.887,-179.977,6.395,149.156
C06088=1140.036,36.929,-50.872,-179.979,6.394,149.157
C06089=1140.041,36.680,-50.858,-179.982,6.393,149.157
C06090=1140.046,36.430,-50.842,-179.985,6.392,149.158
C06091=1140.051,36.180,-50.828,-179.987,6.391,149.158
C06092=1140.057,35.931,-50.812,-179.990,6.390,149.159
C06093=1140.061,35.681,-50.798,-179.992,6.390,149.160
C06094=1140.066,35.432,-50.783,-179.995,6.388,149.160
C06095=1140.072,35.182,-50.768,-179.997,6.387,149.160
C06096=1140.076,34.933,-50.753,180.000,6.386,149.161
C06097=1140.081,34.683,-50.739,179.997,6.385,149.162
C06098=1140.087,34.434,-50.723,179.994,6.384,149.162
C06099=1140.092,34.184,-50.709,179.992,6.383,149.163
C06100=1140.097,33.935,-50.695,179.989,6.381,149.163
C06101=1140.101,33.686,-50.680,179.987,6.381,149.164
C06102=1140.107,33.435,-50.665,179.984,6.380,149.164
C06103=1140.112,33.186,-50.650,179.982,6.378,149.165
C06104=1140.117,32.937,-50.636,179.979,6.378,149.165
C06105=1140.122,32.687,-50.621,179.976,6.376,149.166
C06106=1140.127,32.438,-50.606,179.974,6.375,149.166
C06107=1140.132,32.188,-50.592,179.971,6.375,149.167
C06108=1140.137,31.939,-50.577,179.969,6.373,149.167
C06109=1140.142,31.689,-50.562,179.966,6.373,149.168
C06110=1140.147,31.439,-50.547,179.963,6.371,149.169
C06111=1140.152,31.190,-50.532,179.961,6.370,149.169
C06112=1140.157,30.940,-50.518,179.958,6.369,149.170
C06113=1140.162,30.691,-50.504,179.956,6.368,149.170
C06114=1140.167,30.441,-50.488,179.954,6.368,149.171
C06115=1140.173,30.192,-50.474,179.950,6.366,149.171
C06116=1140.178,29.942,-50.460,179.948,6.365,149.172
C06117=1140.183,29.693,-50.446,179.945,6.364,149.172
C06118=1140.187,29.444,-50.431,179.943,6.363,149.173
C06119=1140.193,29.194,-50.416,179.941,6.363,149.173
C06120=1140.198,28.944,-50.402,179.937,6.361,149.174
C06121=1140.203,28.694,-50.387,179.935,6.361,149.174
C06122=1140.208,28.445,-50.372,179.932,6.359,149.175
C06123=1140.213,28.195,-50.358,179.930,6.358,149.176
C06124=1140.218,27.946,-50.344,179.928,6.358,149.176
C06125=1140.224,27.677,-50.328,179.924,6.356,149.177
C06126=1140.229,27.408,-50.313,179.922,6.356,149.177
C06127=1140.235,27.139,-50.297,179.919,6.354,149.178
C06128=1140.240,26.870,-50.281,179.916,6.353,149.178
C06129=1140.245,26.621,-50.267,179.914,6.352,149.179
C06130=1140.250,26.371,-50.252,179.911,6.351,149.179
C06131=1140.256,26.122,-50.238,179.909,6.350,149.180
C06132=1140.261,25.872,-50.224,179.906,6.349,149.181
C06133=1140.265,25.623,-50.209,179.904,6.349,149.181
C06134=1140.270,25.373,-50.195,179.901,6.347,149.182
C06135=1140.275,25.123,-50.181,179.898,6.346,149.182
C06136=1140.280,24.874,-50.166,179.896,6.345,149.183
C06137=1140.286,24.625,-50.152,179.893,6.344,149.183
C06138=1140.291,24.375,-50.138,179.891,6.344,149.184
C06139=1140.296,24.125,-50.124,179.888,6.342,149.184
C06140=1140.301,23.875,-50.110,179.885,6.342,149.185
C06141=1140.306,23.626,-50.095,179.883,6.341,149.185
C06142=1140.311,23.377,-50.081,179.880,6.339,149.186
C06143=1140.316,23.127,-50.067,179.878,6.339,149.186
C06144=1140.321,22.877,-50.053,179.876,6.338,149.187
C06145=1140.326,22.628,-50.039,179.872,6.337,149.188
C06146=1140.332,22.379,-50.025,179.870,6.336,149.188
C06147=1140.337,22.129,-50.010,179.868,6.335,149.189
C06148=1140.342,21.879,-49.996,179.865,6.334,149.189
C06149=1140.347,21.629,-49.982,179.863,6.333,149.190
C06150=1140.352,21.380,-49.968,179.860,6.332,149.190
C06151=1140.357,21.131,-49.954,179.857,6.331,149.191
C06152=1140.362,20.881,-49.939,179.855,6.330,149.191
C06153=1140.367,20.631,-49.925,179.852,6.330,149.192
C06154=1140.373,20.382,-49.911,179.850,6.328,149.192
C06155=1140.377,20.133,-49.897,179.847,6.327,149.193
C06156=1140.382,19.883,-49.883,179.845,6.327,149.194
C06157=1140.387,19.633,-49.868,179.842,6.325,149.194
C06158=1140.393,19.384,-49.854,179.839,6.325,149.195
C06159=1140.398,19.134,-49.840,179.837,6.324,149.195
C06160=1140.403,18.885,-49.826,179.834,6.322,149.196
C06161=1140.408,18.634,-49.812,179.832,6.322,149.196
C06162=1140.413,18.386,-49.799,179.830,6.321,149.197
C06163=1140.418,18.136,-49.785,179.827,6.319,149.197
C06164=1140.423,17.886,-49.770,179.824,6.319,149.198
C06165=1140.428,17.637,-49.757,179.822,6.318,149.198
C06166=1140.433,17.388,-49.742,179.819,6.317,149.199
C06167=1140.439,17.137,-49.729,179.817,6.316,149.199
C06168=1140.444,16.888,-49.715,179.814,6.315,149.200
C06169=1140.449,16.639,-49.700,179.811,6.314,149.201
C06170=1140.453,16.389,-49.687,179.809,6.313,149.201
C06171=1140.459,16.140,-49.673,179.806,6.313,149.202
C06172=1140.464,15.890,-49.659,179.804,6.311,149.202
C06173=1140.469,15.640,-49.645,179.801,6.310,149.203
C06174=1140.475,15.391,-49.631,179.799,6.310,149.203
C06175=1140.479,15.142,-49.617,179.797,6.309,149.204
C06176=1140.484,14.891,-49.604,179.794,6.307,149.204
C06177=1140.490,14.642,-49.590,179.791,6.307,149.205
C06178=1140.495,14.393,-49.576,179.789,6.306,149.205
C06179=1140.500,14.143,-49.561,179.786,6.305,149.206
C06180=1140.505,13.894,-49.549,179.784,6.304,149.207
C06181=1140.510,13.644,-49.535,179.781,6.303,149.207
C06182=1140.515,13.395,-49.521,179.778,6.302,149.208
C06183=1140.520,13.145,-49.507,179.776,6.301,149.208
C06184=1140.525,12.895,-49.493,179.773,6.301,149.209
C06185=1140.530,12.646,-49.479,179.771,6.300,149.209
C06186=1140.536,12.396,-49.466,179.768,6.298,149.210
C06187=1140.541,12.147,-49.452,179.766,6.298,149.210
C06188=1140.546,11.897,-49.438,179.764,6.297,149.211
C06189=1140.551,11.647,-49.425,179.761,6.296,149.211
C06190=1140.556,11.398,-49.411,179.758,6.295,149.212
C06191=1140.561,11.148,-49.397,179.756,6.294,149.213
C06192=1140.566,10.899,-49.384,179.753,6.294,149.213
C06193=1140.571,10.649,-49.370,179.750,6.292,149.214
C06194=1140.576,10.399,-49.356,179.748,6.291,149.214
C06195=1140.582,10.150,-49.342,179.746,6.291,149.215
C06196=1140.586,9.900,-49.329,179.744,6.290,149.215
C06197=1140.592,9.651,-49.315,179.740,6.289,149.216
C06198=1140.597,9.401,-49.302,179.738,6.288,149.216
C06199=1140.602,9.152,-49.288,179.736,6.287,149.217
C06200=1140.607,8.902,-49.274,179.733,6.287,149.218
C06201=1140.613,8.653,-49.261,179.730,6.285,149.218
C06202=1140.617,8.403,-49.247,179.728,6.285,149.219
C06203=1140.623,8.154,-49.234,179.726,6.284,149.219
C06204=1140.627,7.904,-49.220,179.723,6.283,149.220
C06205=1140.633,7.655,-49.207,179.720,6.282,149.220
C06206=1140.638,7.404,-49.194,179.718,6.281,149.221
C06207=1140.643,7.155,-49.180,179.716,6.280,149.221
C06208=1140.648,6.905,-49.167,179.713,6.280,149.222
C06209=1140.653,6.655,-49.153,179.710,6.278,149.222
C06210=1140.659,6.406,-49.140,179.708,6.278,149.223
C06211=1140.663,6.156,-49.126,179.706,6.277,149.224
C06212=1140.669,5.907,-49.113,179.703,6.276,149.224
C06213=1140.674,5.657,-49.099,179.700,6.275,149.225
C06214=1140.679,5.408,-49.086,179.698,6.274,149.225
C06215=1140.684,5.158,-49.073,179.695,6.274,149.226
C06216=1140.689,4.909,-49.059,179.693,6.273,149.226
C06217=1140.695,4.659,-49.046,179.690,6.271,149.227
C06218=1140.700,4.409,-49.033,179.688,6.271,149.227
C06219=1140.705,4.160,-49.019,179.686,6.270,149.228
C06220=1140.710,3.910,-49.006,179.683,6.270,149.229
C06221=1140.715,3.661,-48.992,179.681,6.269,149.229
C06222=1140.720,3.411,-48.979,179.678,6.267,149.230
C06223=1140.725,3.162,-48.966,179.675,6.267,149.230
C06224=1140.730,2.912,-48.952,179.673,6.266,149.231
C06225=1140.735,2.663,-48.939,179.670,6.266,149.231
C06226=1140.740,2.412,-48.926,179.668,6.264,149.232
C06227=1140.746,2.163,-48.913,179.666,6.263,149.232
C06228=1140.751,1.914,-48.899,179.663,6.263,149.233
C06229=1140.756,1.644,-48.886,179.661,6.262,149.233
C06230=1140.762,1.375,-48.871,179.657,6.261,149.234
C06231=1140.767,1.105,-48.856,179.655,6.260,149.235
C06232=1140.773,0.836,-48.843,179.652,6.259,149.235
C06233=1140.778,0.586,-48.829,179.650,6.258,149.236
C06234=1140.783,0.337,-48.816,179.647,6.257,149.236
C06235=1140.789,0.087,-48.803,179.645,6.257,149.237
C06236=1140.793,-0.163,-48.790,179.642,6.256,149.238
C06237=1140.799,-0.412,-48.777,179.640,6.255,149.238
C06238=1140.803,-0.662,-48.763,179.637,6.254,149.239
C06239=1140.809,-0.912,-48.750,179.635,6.253,149.239
C06240=1140.814,-1.161,-48.737,179.633,6.253,149.240
C06241=1140.819,-1.411,-48.724,179.630,6.252,149.240
C06242=1140.825,-1.660,-48.711,179.628,6.251,149.241
C06243=1140.830,-1.910,-48.698,179.625,6.250,149.241
C06244=1140.835,-2.160,-48.684,179.622,6.249,149.242
C06245=1140.840,-2.409,-48.672,179.620,6.249,149.242
C06246=1140.845,-2.659,-48.659,179.618,6.248,149.243
C06247=1140.850,-2.908,-48.645,179.615,6.247,149.244
C06248=1140.856,-3.158,-48.633,179.613,6.246,149.244
C06249=1140.860,-3.408,-48.620,179.610,6.245,149.245
C06250=1140.866,-3.657,-48.607,179.608,6.244,149.245
C06251=1140.871,-3.907,-48.594,179.606,6.244,149.246
C06252=1140.876,-4.157,-48.581,179.603,6.243,149.246
C06253=1140.881,-4.406,-48.568,179.601,6.242,149.247
C06254=1140.886,-4.655,-48.555,179.597,6.241,149.248
C06255=1140.891,-4.905,-48.542,179.595,6.240,149.248
C06256=1140.897,-5.155,-48.528,179.593,6.240,149.249
C06257=1140.902,-5.404,-48.516,179.590,6.239,149.249
C06258=1140.907,-5.653,-48.503,179.588,6.238,149.250
C06259=1140.912,-5.904,-48.490,179.586,6.238,149.250
C06260=1140.917,-6.153,-48.477,179.583,6.236,149.251
C06261=1140.922,-6.402,-48.464,179.581,6.236,149.251
C06262=1140.928,-6.653,-48.451,179.578,6.235,149.252
C06263=1140.933,-6.902,-48.438,179.576,6.234,149.252
C06264=1140.938,-7.151,-48.426,179.573,6.234,149.253
C06265=1140.943,-7.401,-48.413,179.571,6.233,149.254
C06266=1140.948,-7.651,-48.400,179.568,6.231,149.254
C06267=1140.954,-7.901,-48.388,179.565,6.231,149.255
C06268=1140.959,-8.150,-48.375,179.563,6.230,149.255
C06269=1140.963,-8.400,-48.362,179.561,6.229,149.256
C06270=1140.969,-8.650,-48.349,179.558,6.229,149.256
C06271=1140.974,-8.899,-48.336,179.556,6.228,149.257
C06272=1140.980,-9.148,-48.324,179.554,6.228,149.258
C06273=1140.984,-9.399,-48.311,179.551,6.226,149.258
C06274=1140.989,-9.648,-48.298,179.549,6.225,149.258
C06275=1140.995,-9.897,-48.285,179.546,6.225,149.259
C06276=1141.000,-10.147,-48.272,179.544,6.224,149.260
C06277=1141.005,-10.397,-48.259,179.541,6.224,149.260
C06278=1141.010,-10.647,-48.247,179.539,6.223,149.261
C06279=1141.015,-10.896,-48.235,179.537,6.222,149.261
C06280=1141.020,-11.145,-48.222,179.534,6.222,149.262
C06281=1141.026,-11.395,-48.209,179.531,6.220,149.262
C06282=1141.031,-11.645,-48.196,179.529,6.220,149.263
C06283=1141.036,-11.895,-48.184,179.527,6.219,149.264
C06284=1141.041,-12.144,-48.172,179.524,6.218,149.264
C06285=1141.046,-12.394,-48.159,179.522,6.218,149.265
C06286=1141.052,-12.643,-48.146,179.520,6.217,149.265
C06287=1141.056,-12.893,-48.133,179.517,6.217,149.266
C06288=1141.062,-13.143,-48.121,179.515,6.216,149.266
C06289=1141.067,-13.392,-48.108,179.512,6.214,149.267
C06290=1141.072,-13.642,-48.096,179.509,6.214,149.268
C06291=1141.078,-13.891,-48.083,179.507,6.213,149.268
C06292=1141.082,-14.142,-48.071,179.505,6.212,149.269
C06293=1141.088,-14.391,-48.058,179.502,6.212,149.269
C06294=1141.093,-14.640,-48.046,179.500,6.211,149.270
C06295=1141.098,-14.890,-48.033,179.497,6.210,149.270
C06296=1141.103,-15.140,-48.021,179.495,6.210,149.271
C06297=1141.108,-15.389,-48.009,179.493,6.209,149.271
C06298=1141.113,-15.639,-47.996,179.490,6.208,149.272
C06299=1141.119,-15.889,-47.983,179.488,6.207,149.272
C06300=1141.124,-16.139,-47.971,179.485,6.206,149.273
C06301=1141.129,-16.388,-47.958,179.483,6.206,149.274
C06302=1141.135,-16.638,-47.946,179.481,6.205,149.274
C06303=1141.140,-16.887,-47.934,179.478,6.204,149.275
C06304=1141.145,-17.136,-47.921,179.476,6.204,149.275
C06305=1141.150,-17.386,-47.909,179.474,6.203,149.276
C06306=1141.155,-17.636,-47.896,179.471,6.202,149.276
C06307=1141.160,-17.886,-47.884,179.469,6.202,149.277
C06308=1141.165,-18.136,-47.872,179.466,6.201,149.278
C06309=1141.171,-18.385,-47.859,179.464,6.200,149.278
C06310=1141.176,-18.635,-47.847,179.461,6.199,149.279
C06311=1141.181,-18.884,-47.834,179.458,6.198,149.279
C06312=1141.187,-19.134,-47.823,179.456,6.198,149.280
C06313=1141.192,-19.383,-47.810,179.454,6.197,149.280
C06314=1141.197,-19.633,-47.798,179.451,6.196,149.281
C06315=1141.202,-19.883,-47.786,179.449,6.196,149.281
C06316=1141.207,-20.132,-47.773,179.447,6.195,149.282
C06317=1141.212,-20.383,-47.761,179.444,6.194,149.283
C06318=1141.217,-20.632,-47.748,179.442,6.194,149.283
C06319=1141.223,-20.882,-47.736,179.440,6.193,149.284
C06320=1141.227,-21.131,-47.724,179.437,6.192,149.284
C06321=1141.233,-21.381,-47.712,179.435,6.192,149.285
C06322=1141.238,-21.630,-47.700,179.433,6.191,149.285
C06323=1141.243,-21.880,-47.688,179.430,6.190,149.286
C06324=1141.248,-22.129,-47.675,179.428,6.190,149.286
C06325=1141.254,-22.379,-47.663,179.425,6.188,149.287
C06326=1141.259,-22.629,-47.651,179.423,6.188,149.287
C06327=1141.264,-22.879,-47.639,179.420,6.187,149.288
C06328=1141.270,-23.129,-47.627,179.418,6.186,149.289
C06329=1141.275,-23.378,-47.614,179.415,6.186,149.289
C06330=1141.280,-23.628,-47.602,179.413,6.185,149.290
C06331=1141.285,-23.877,-47.590,179.411,6.184,149.290
C06332=1141.290,-24.127,-47.579,179.408,6.184,149.291
C06333=1141.296,-24.397,-47.565,179.406,6.183,149.291
C06334=1141.302,-24.667,-47.552,179.403,6.183,149.292
C06335=1141.307,-24.937,-47.539,179.401,6.181,149.293
C06336=1141.312,-25.207,-47.526,179.398,6.181,149.293
C06337=1141.318,-25.457,-47.514,179.396,6.180,149.294
C06338=1141.323,-25.707,-47.502,179.393,6.180,149.294
C06339=1141.328,-25.956,-47.489,179.391,6.179,149.295
C06340=1141.333,-26.206,-47.478,179.388,6.178,149.296
C06341=1141.339,-26.455,-47.467,179.386,6.178,149.296
C06342=1141.344,-26.705,-47.454,179.384,6.177,149.297
C06343=1141.350,-26.954,-47.442,179.381,6.176,149.297
C06344=1141.355,-27.204,-47.430,179.379,6.176,149.298
C06345=1141.359,-27.453,-47.418,179.377,6.175,149.298
C06346=1141.365,-27.703,-47.406,179.374,6.174,149.299
C06347=1141.370,-27.953,-47.394,179.372,6.174,149.299
C06348=1141.375,-28.203,-47.382,179.369,6.173,149.300
C06349=1141.380,-28.452,-47.371,179.367,6.172,149.301
C06350=1141.385,-28.702,-47.359,179.365,6.172,149.301
C06351=1141.391,-28.952,-47.347,179.362,6.171,149.302
C06352=1141.396,-29.201,-47.334,179.360,6.170,149.302
C06353=1141.401,-29.451,-47.323,179.358,6.170,149.303
C06354=1141.406,-29.701,-47.311,179.355,6.169,149.303
C06355=1141.412,-29.951,-47.299,179.353,6.169,149.304
C06356=1141.417,-30.201,-47.287,179.350,6.168,149.305
C06357=1141.421,-30.450,-47.275,179.348,6.167,149.305
C06358=1141.427,-30.700,-47.263,179.346,6.167,149.305
C06359=1141.433,-30.949,-47.252,179.343,6.166,149.306
C06360=1141.438,-31.199,-47.240,179.341,6.165,149.307
C06361=1141.443,-31.449,-47.229,179.339,6.165,149.307
C06362=1141.448,-31.698,-47.216,179.336,6.164,149.308
C06363=1141.454,-31.948,-47.204,179.334,6.163,149.308
C06364=1141.458,-32.197,-47.193,179.331,6.163,149.309
C06365=1141.464,-32.447,-47.181,179.329,6.162,149.309
C06366=1141.469,-32.697,-47.169,179.327,6.161,149.310
C06367=1141.474,-32.947,-47.158,179.324,6.161,149.311
C06368=1141.480,-33.196,-47.146,179.322,6.160,149.311
C06369=1141.485,-33.446,-47.134,179.320,6.159,149.312
C06370=1141.490,-33.695,-47.122,179.317,6.159,149.312
C06371=1141.495,-33.945,-47.111,179.315,6.158,149.313
C06372=1141.500,-34.195,-47.099,179.313,6.157,149.313
C06373=1141.505,-34.445,-47.087,179.310,6.157,149.314
C06374=1141.511,-34.695,-47.075,179.308,6.156,149.314
C06375=1141.516,-34.944,-47.065,179.305,6.156,149.315
C06376=1141.521,-35.193,-47.053,179.303,6.155,149.316
C06377=1141.527,-35.443,-47.041,179.301,6.154,149.316
C06378=1141.531,-35.693,-47.029,179.298,6.154,149.317
C06379=1141.537,-35.943,-47.018,179.296,6.153,149.317
C06380=1141.542,-36.193,-47.006,179.294,6.152,149.318
C06381=1141.548,-36.442,-46.995,179.291,6.152,149.318
C06382=1141.553,-36.692,-46.983,179.289,6.151,149.319
C06383=1141.558,-36.941,-46.972,179.287,6.150,149.319
C06384=1141.563,-37.191,-46.960,179.284,6.150,149.320
C06385=1141.568,-37.441,-46.948,179.282,6.149,149.321
C06386=1141.574,-37.690,-46.937,179.280,6.149,149.321
C06387=1141.579,-37.940,-46.925,179.277,6.148,149.322
C06388=1141.584,-38.190,-46.914,179.275,6.147,149.322
C06389=1141.589,-38.440,-46.902,179.272,6.147,149.323
C06390=1141.594,-38.689,-46.891,179.270,6.146,149.323
C06391=1141.600,-38.939,-46.879,179.268,6.145,149.324
C06392=1141.605,-39.188,-46.868,179.265,6.145,149.325
C06393=1141.610,-39.438,-46.856,179.263,6.144,149.325
C06394=1141.615,-39.688,-46.845,179.262,6.144,149.325
C06395=1141.621,-39.938,-46.834,179.259,6.144,149.326
C06396=1141.626,-40.187,-46.822,179.257,6.143,149.327
C06397=1141.631,-40.437,-46.811,179.255,6.142,149.327
C06398=1141.636,-40.687,-46.799,179.252,6.142,149.328
C06399=1141.642,-40.937,-46.787,179.250,6.141,149.328
C06400=1141.647,-41.186,-46.776,179.247,6.140,149.329
C06401=1141.652,-41.436,-46.765,179.245,6.140,149.329
C06402=1141.657,-41.685,-46.753,179.243,6.139,149.330
C06403=1141.663,-41.936,-46.742,179.240,6.139,149.331
C06404=1141.668,-42.185,-46.731,179.238,6.138,149.331
C06405=1141.673,-42.435,-46.719,179.236,6.137,149.332
C06406=1141.678,-42.684,-46.708,179.233,6.137,149.332
C06407=1141.683,-42.933,-46.697,179.231,6.136,149.333
C06408=1141.689,-43.184,-46.686,179.229,6.135,149.333
C06409=1141.694,-43.433,-46.675,179.226,6.135,149.334
C06410=1141.699,-43.683,-46.663,179.224,6.134,149.334
C06411=1141.705,-43.932,-46.652,179.222,6.134,149.335
C06412=1141.710,-44.182,-46.640,179.220,6.133,149.336
C06413=1141.715,-44.432,-46.629,179.217,6.133,149.336
C06414=1141.720,-44.681,-46.618,179.215,6.132,149.337
C06415=1141.726,-44.931,-46.607,179.213,6.131,149.337
C06416=1141.730,-45.181,-46.595,179.210,6.131,149.338
C06417=1141.736,-45.431,-46.584,179.208,6.130,149.338
C06418=1141.741,-45.680,-46.573,179.205,6.130,149.339
C06419=1141.746,-45.930,-46.562,179.203,6.129,149.339
C06420=1141.752,-46.180,-46.550,179.201,6.128,149.340
C06421=1141.757,-46.429,-46.540,179.198,6.128,149.341
C06422=1141.762,-46.679,-46.529,179.196,6.127,149.341
C06423=1141.767,-46.929,-46.517,179.195,6.127,149.342
C06424=1141.773,-47.179,-46.506,179.192,6.126,149.342
C06425=1141.778,-47.428,-46.495,179.190,6.126,149.343
C06426=1141.783,-47.678,-46.483,179.187,6.125,149.343
C06427=1141.789,-47.928,-46.473,179.185,6.124,149.344
C06428=1141.794,-48.178,-46.461,179.183,6.124,149.344
C06429=1141.799,-48.427,-46.450,179.180,6.123,149.345
C06430=1141.804,-48.677,-46.440,179.178,6.122,149.346
C06431=1141.809,-48.926,-46.428,179.176,6.122,149.346
C06432=1141.815,-49.176,-46.418,179.173,6.121,149.347
C06433=1141.820,-49.426,-46.406,179.171,6.121,149.347
C06434=1141.825,-49.675,-46.395,179.169,6.121,149.348
C06435=1141.831,-49.925,-46.384,179.167,6.120,149.348
C06436=1141.836,-50.175,-46.373,179.164,6.119,149.349
C06437=1141.842,-50.445,-46.361,179.162,6.119,149.349
C06438=1141.848,-50.716,-46.349,179.160,6.118,149.350
C06439=1141.852,-50.987,-46.337,179.157,6.117,149.351
C06440=1141.859,-51.258,-46.326,179.155,6.117,149.351
C06441=1141.864,-51.507,-46.315,179.152,6.116,149.352
C06442=1141.869,-51.757,-46.303,179.150,6.116,149.352
C06443=1141.875,-52.007,-46.293,179.148,6.115,149.353
C06444=1141.879,-52.257,-46.281,179.145,6.114,149.353
C06445=1141.885,-52.506,-46.271,179.143,6.114,149.354
C06446=1141.890,-52.756,-46.259,179.141,6.113,149.355
C06447=1141.895,-53.006,-46.249,179.138,6.112,149.355
C06448=1141.901,-53.255,-46.238,179.136,6.113,149.356
C06449=1141.906,-53.505,-46.227,179.134,6.112,149.356
C06450=1141.911,-53.754,-46.216,179.132,6.111,149.357
C06451=1141.917,-54.005,-46.205,179.129,6.111,149.357
C06452=1141.922,-54.254,-46.194,179.127,6.110,149.358
C06453=1141.927,-54.504,-46.183,179.125,6.109,149.358
C06454=1141.932,-54.753,-46.173,179.122,6.109,149.359
C06455=1141.937,-55.003,-46.162,179.120,6.108,149.360
C06456=1141.943,-55.254,-46.151,179.118,6.108,149.360
C06457=1141.948,-55.503,-46.140,179.116,6.108,149.361
C06458=1141.953,-55.753,-46.129,179.114,6.107,149.361
C06459=1141.959,-56.002,-46.118,179.111,6.106,149.362
C06460=1141.964,-56.252,-46.108,179.109,6.105,149.362
C06461=1141.969,-56.502,-46.098,179.107,6.105,149.363
C06462=1141.974,-56.751,-46.086,179.104,6.104,149.363
C06463=1141.979,-57.001,-46.076,179.103,6.104,149.364
C06464=1141.985,-57.251,-46.064,179.100,6.104,149.365
C06465=1141.991,-57.500,-46.054,179.098,6.103,149.365
C06466=1141.996,-57.751,-46.043,179.096,6.102,149.366
C06467=1142.001,-57.999,-46.033,179.093,6.102,149.366
C06468=1142.006,-58.250,-46.022,179.091,6.101,149.367
C06469=1142.011,-58.499,-46.012,179.089,6.101,149.367
C06470=1142.016,-58.749,-46.000,179.087,6.101,149.368
C06471=1142.022,-58.998,-45.990,179.084,6.100,149.368
C06472=1142.027,-59.249,-45.980,179.082,6.099,149.369
C06473=1142.032,-59.498,-45.969,179.080,6.099,149.370
C06474=1142.038,-59.748,-45.958,179.077,6.098,149.370
C06475=1142.043,-59.998,-45.947,179.075,6.097,149.371
C06476=1142.048,-60.247,-45.936,179.074,6.097,149.371
C06477=1142.054,-60.497,-45.926,179.071,6.097,149.372
C06478=1142.059,-60.747,-45.915,179.069,6.096,149.372
C06479=1142.064,-60.997,-45.905,179.067,6.095,149.373
C06480=1142.069,-61.246,-45.894,179.064,6.095,149.373
C06481=1142.074,-61.496,-45.884,179.062,6.095,149.374
C06482=1142.079,-61.746,-45.873,179.060,6.094,149.374
C06483=1142.085,-61.996,-45.863,179.057,6.094,149.375
C06484=1142.090,-62.245,-45.852,179.055,6.093,149.376
C06485=1142.095,-62.495,-45.841,179.053,6.092,149.376
C06486=1142.101,-62.744,-45.831,179.050,6.092,149.377
C06487=1142.106,-62.995,-45.821,179.049,6.092,149.377
C06488=1142.111,-63.244,-45.810,179.047,6.091,149.378
C06489=1142.116,-63.494,-45.799,179.044,6.090,149.378
C06490=1142.122,-63.743,-45.789,179.042,6.090,149.379
C06491=1142.127,-63.994,-45.778,179.040,6.089,149.379
C06492=1142.132,-64.243,-45.768,179.037,6.089,149.380
C06493=1142.138,-64.493,-45.758,179.035,6.089,149.381
C06494=1142.143,-64.742,-45.747,179.033,6.088,149.381
C06495=1142.148,-64.992,-45.736,179.031,6.087,149.381
C06496=1142.153,-65.242,-45.726,179.028,6.087,149.382
C06497=1142.159,-65.492,-45.716,179.026,6.086,149.383
C06498=1142.165,-65.741,-45.705,179.024,6.086,149.383
C06499=1142.170,-65.991,-45.695,179.022,6.086,149.384
C06500=1142.175,-66.241,-45.685,179.020,6.085,149.384
C06501=1142.180,-66.491,-45.674,179.017,6.084,149.385
C06502=1142.185,-66.740,-45.663,179.015,6.084,149.385
C06503=1142.190,-66.989,-45.653,179.013,6.084,149.386
C06504=1142.195,-67.240,-45.643,179.011,6.083,149.386
C06505=1142.201,-67.489,-45.633,179.009,6.082,149.387
C06506=1142.206,-67.739,-45.622,179.007,6.082,149.387
C06507=1142.211,-67.989,-45.612,179.004,6.081,149.388
C06508=1142.217,-68.238,-45.602,179.002,6.081,149.389
C06509=1142.222,-68.489,-45.591,179.000,6.081,149.389
C06510=1142.228,-68.738,-45.581,178.997,6.080,149.390
C06511=1142.233,-68.988,-45.571,178.995,6.079,149.390
C06512=1142.238,-69.238,-45.560,178.993,6.079,149.391
C06513=1142.243,-69.487,-45.550,178.991,6.079,149.391
C06514=1142.249,-69.737,-45.540,178.989,6.078,149.392
C06515=1142.254,-69.987,-45.530,178.987,6.078,149.392
C06516=1142.259,-70.237,-45.519,178.984,6.077,149.393
C06517=1142.265,-70.486,-45.509,178.983,6.077,149.393
C06518=1142.270,-70.736,-45.499,178.980,6.076,149.394
C06519=1142.276,-70.986,-45.488,178.978,6.076,149.395
C06520=1142.280,-71.235,-45.479,178.976,6.075,149.395
C06521=1142.286,-71.485,-45.469,178.973,6.075,149.396
C06522=1142.291,-71.735,-45.458,178.971,6.075,149.396
C06523=1142.297,-71.984,-45.448,178.969,6.074,149.397
C06524=1142.302,-72.234,-45.438,178.967,6.073,149.397
C06525=1142.307,-72.484,-45.427,178.964,6.073,149.398
C06526=1142.312,-72.733,-45.417,178.963,6.073,149.398
C06527=1142.318,-72.983,-45.407,178.961,6.072,149.399
C06528=1142.323,-73.233,-45.397,178.958,6.071,149.399
C06529=1142.329,-73.483,-45.387,178.956,6.071,149.400
C06530=1142.334,-73.733,-45.377,178.954,6.071,149.401
C06531=1142.339,-73.982,-45.367,178.952,6.070,149.401
C06532=1142.344,-74.232,-45.357,178.949,6.070,149.402
C06533=1142.350,-74.482,-45.347,178.947,6.069,149.402
C06534=1142.355,-74.732,-45.336,178.946,6.069,149.403
C06535=1142.361,-74.981,-45.326,178.943,6.068,149.403
C06536=1142.365,-75.231,-45.316,178.941,6.068,149.404
C06537=1142.371,-75.481,-45.307,178.938,6.067,149.404
C06538=1142.377,-75.731,-45.297,178.937,6.067,149.405
C06539=1142.382,-75.980,-45.286,178.935,6.066,149.405
C06540=1142.386,-76.230,-45.276,178.932,6.066,149.406
C06541=1142.393,-76.501,-45.265,178.930,6.065,149.407
C06542=1142.398,-76.773,-45.255,178.928,6.064,149.407
C06543=1142.404,-77.045,-45.243,178.925,6.064,149.408
C06544=1142.410,-77.315,-45.233,178.923,6.063,149.408
C06545=1142.415,-77.566,-45.223,178.921,6.064,149.409
C06546=1142.421,-77.816,-45.213,178.918,6.063,149.409
C06547=1142.426,-78.065,-45.203,178.916,6.062,149.410
C06548=1142.431,-78.314,-45.193,178.914,6.061,149.410
C06549=1142.437,-78.565,-45.183,178.912,6.062,149.411
C06550=1142.442,-78.815,-45.173,178.910,6.061,149.412
C06551=1142.447,-79.064,-45.163,178.908,6.060,149.412
C06552=1142.453,-79.314,-45.153,178.906,6.060,149.413
C06553=1142.458,-79.563,-45.144,178.903,6.060,149.413
C06554=1142.464,-79.813,-45.134,178.901,6.059,149.414
C06555=1142.469,-80.063,-45.123,178.899,6.058,149.414
C06556=1142.473,-80.312,-45.114,178.897,6.058,149.415
C06557=1142.479,-80.563,-45.104,178.895,6.058,149.415
C06558=1142.485,-80.812,-45.094,178.893,6.057,149.416
C06559=1142.490,-81.061,-45.084,178.890,6.056,149.416
C06560=1142.495,-81.312,-45.075,178.889,6.056,149.417
C06561=1142.501,-81.562,-45.064,178.886,6.056,149.418
C06562=1142.506,-81.811,-45.055,178.884,6.055,149.418
C06563=1142.512,-82.061,-45.045,178.882,6.055,149.419
C06564=1142.516,-82.310,-45.036,178.880,6.055,149.419
C06565=1142.522,-82.560,-45.025,178.878,6.054,149.420
C06566=1142.527,-82.811,-45.016,178.875,6.053,149.420
C06567=1142.532,-83.060,-45.006,178.874,6.054,149.421
C06568=1142.538,-83.310,-44.996,178.871,6.053,149.421
C06569=1142.543,-83.559,-44.987,178.869,6.052,149.422
C06570=1142.548,-83.809,-44.977,178.867,6.052,149.422
C06571=1142.554,-84.059,-44.967,178.865,6.052,149.423
C06572=1142.559,-84.308,-44.958,178.863,6.051,149.423
C06573=1142.564,-84.559,-44.947,178.861,6.050,149.424
C06574=1142.569,-84.809,-44.938,178.859,6.051,149.425
C06575=1142.575,-85.058,-44.928,178.856,6.050,149.425
C06576=1142.580,-85.308,-44.919,178.854,6.049,149.426
C06577=1142.586,-85.557,-44.909,178.853,6.049,149.426
C06578=1142.591,-85.807,-44.900,178.850,6.048,149.426
C06579=1142.597,-86.057,-44.890,178.848,6.048,149.427
C06580=1142.601,-86.307,-44.880,178.846,6.048,149.428
C06581=1142.607,-86.557,-44.870,178.844,6.047,149.428
C06582=1142.612,-86.806,-44.860,178.842,6.046,149.429
C06583=1142.617,-87.056,-44.851,178.839,6.046,149.429
C06584=1142.623,-87.306,-44.841,178.837,6.046,149.430
C06585=1142.628,-87.556,-44.832,178.835,6.045,149.430
C06586=1142.634,-87.805,-44.822,178.833,6.045,149.431
C06587=1142.639,-88.055,-44.813,178.831,6.045,149.431
C06588=1142.645,-88.305,-44.803,178.829,6.044,149.432
C06589=1142.650,-88.555,-44.794,178.827,6.043,149.432
C06590=1142.655,-88.804,-44.784,178.825,6.044,149.433
C06591=1142.660,-89.055,-44.774,178.823,6.043,149.433
C06592=1142.665,-89.304,-44.765,178.821,6.042,149.434
C06593=1142.671,-89.554,-44.755,178.819,6.042,149.435
C06594=1142.676,-89.803,-44.746,178.816,6.042,149.435
C06595=1142.681,-90.053,-44.736,178.814,6.041,149.436
C06596=1142.687,-90.303,-44.727,178.813,6.041,149.436
C06597=1142.692,-90.553,-44.717,178.810,6.040,149.437
C06598=1142.697,-90.803,-44.708,178.808,6.040,149.437
C06599=1142.703,-91.052,-44.698,178.806,6.040,149.438
C06600=1142.708,-91.302,-44.689,178.804,6.039,149.438
C06601=1142.713,-91.551,-44.679,178.802,6.038,149.439
C06602=1142.719,-91.801,-44.670,178.799,6.038,149.439
C06603=1142.724,-92.051,-44.661,178.797,6.038,149.440
C06604=1142.730,-92.301,-44.651,178.795,6.037,149.440
C06605=1142.735,-92.551,-44.642,178.793,6.036,149.441
C06606=1142.741,-92.801,-44.632,178.791,6.037,149.441
C06607=1142.746,-93.050,-44.623,178.789,6.036,149.442
C06608=1142.751,-93.300,-44.614,178.787,6.036,149.443
C06609=1142.756,-93.549,-44.604,178.785,6.035,149.443
C06610=1142.762,-93.799,-44.595,178.783,6.035,149.444
C06611=1142.767,-94.049,-44.585,178.781,6.035,149.444
C06612=1142.772,-94.299,-44.576,178.779,6.034,149.445
C06613=1142.777,-94.549,-44.567,178.777,6.033,149.445
C06614=1142.783,-94.799,-44.557,178.775,6.034,149.446
C06615=1142.789,-95.049,-44.548,178.773,6.033,149.446
C06616=1142.793,-95.298,-44.539,178.770,6.032,149.447
C06617=1142.799,-95.548,-44.529,178.769,6.032,149.447
C06618=1142.804,-95.798,-44.520,178.767,6.031,149.448
C06619=1142.809,-96.047,-44.511,178.764,6.031,149.448
C06620=1142.815,-96.297,-44.501,178.762,6.031,149.449
C06621=1142.820,-96.547,-44.492,178.760,6.030,149.449
C06622=1142.826,-96.797,-44.483,178.758,6.030,149.450
C06623=1142.831,-97.046,-44.473,178.756,6.030,149.450
C06624=1142.836,-97.296,-44.464,178.754,6.029,149.451
C06625=1142.842,-97.546,-44.455,178.751,6.028,149.452
C06626=1142.847,-97.796,-44.446,178.750,6.028,149.452
C06627=1142.852,-98.046,-44.436,178.748,6.028,149.452
C06628=1142.857,-98.295,-44.427,178.746,6.028,149.453
C06629=1142.863,-98.546,-44.418,178.744,6.027,149.453
C06630=1142.869,-98.795,-44.409,178.742,6.026,149.454
C06631=1142.874,-99.045,-44.400,178.740,6.027,149.455
C06632=1142.879,-99.295,-44.390,178.737,6.026,149.455
C06633=1142.884,-99.545,-44.381,178.735,6.025,149.456
C06634=1142.890,-99.794,-44.372,178.734,6.025,149.456
C06635=1142.895,-100.044,-44.364,178.731,6.024,149.457
C06636=1142.901,-100.294,-44.354,178.729,6.024,149.457
C06637=1142.906,-100.543,-44.344,178.727,6.024,149.458
C06638=1142.911,-100.793,-44.336,178.725,6.023,149.458
C06639=1142.916,-101.043,-44.327,178.723,6.023,149.459
C06640=1142.922,-101.293,-44.317,178.721,6.023,149.459
C06641=1142.928,-101.543,-44.308,178.719,6.022,149.460
C06642=1142.933,-101.793,-44.299,178.717,6.022,149.460
C06643=1142.938,-102.043,-44.291,178.715,6.021,149.461
C06644=1142.943,-102.292,-44.280,178.712,6.021,149.461
C06645=1142.949,-102.565,-44.271,178.711,6.021,149.462
C06646=1142.955,-102.836,-44.261,178.709,6.020,149.462
C06647=1142.961,-103.108,-44.251,178.706,6.020,149.463
C06648=1142.967,-103.381,-44.242,178.704,6.019,149.464
C06649=1142.972,-103.630,-44.232,178.702,6.019,149.464
C06650=1142.977,-103.880,-44.223,178.700,6.018,149.465
C06651=1142.983,-104.130,-44.214,178.698,6.018,149.465
C06652=1142.988,-104.380,-44.205,178.696,6.018,149.466
C06653=1142.994,-104.629,-44.196,178.693,6.017,149.466
C06654=1142.999,-104.879,-44.188,178.692,6.017,149.467
C06655=1143.004,-105.129,-44.179,178.690,6.017,149.467
C06656=1143.009,-105.379,-44.170,178.688,6.017,149.468
C06657=1143.015,-105.629,-44.160,178.686,6.016,149.468
C06658=1143.020,-105.879,-44.151,178.684,6.015,149.469
C06659=1143.026,-106.129,-44.142,178.682,6.015,149.469
C06660=1143.031,-106.378,-44.134,178.679,6.015,149.470
C06661=1143.037,-106.628,-44.125,178.678,6.015,149.470
C06662=1143.042,-106.877,-44.116,178.676,6.014,149.471
C06663=1143.047,-107.127,-44.107,178.673,6.013,149.471
C06664=1143.052,-107.377,-44.098,178.672,6.013,149.472
C06665=1143.058,-107.627,-44.089,178.670,6.013,149.472
C06666=1143.064,-107.876,-44.080,178.668,6.013,149.473
C06667=1143.069,-108.126,-44.071,178.666,6.012,149.473
C06668=1143.074,-108.376,-44.063,178.663,6.011,149.474
C06669=1143.079,-108.626,-44.054,178.662,6.012,149.474
C06670=1143.084,-108.876,-44.045,178.659,6.011,149.475
C06671=1143.090,-109.126,-44.036,178.658,6.011,149.475
C06672=1143.095,-109.375,-44.027,178.656,6.010,149.476
C06673=1143.100,-109.625,-44.018,178.653,6.009,149.476
C06674=1143.106,-109.875,-44.009,178.652,6.009,149.477
C06675=1143.112,-110.125,-44.001,178.650,6.009,149.477
C06676=1143.117,-110.375,-43.992,178.648,6.009,149.478
C06677=1143.123,-110.624,-43.983,178.645,6.008,149.479
C06678=1143.128,-110.874,-43.974,178.644,6.008,149.479
C06679=1143.133,-111.124,-43.966,178.642,6.008,149.480
C06680=1143.138,-111.374,-43.957,178.639,6.007,149.480
C06681=1143.143,-111.624,-43.948,178.638,6.007,149.481
C06682=1143.149,-111.873,-43.939,178.636,6.006,149.481
C06683=1143.154,-112.123,-43.930,178.634,6.006,149.482
C06684=1143.160,-112.373,-43.922,178.632,6.005,149.482
C06685=1143.165,-112.623,-43.913,178.630,6.005,149.482
C06686=1143.171,-112.872,-43.905,178.628,6.005,149.483
C06687=1143.176,-113.122,-43.896,178.625,6.004,149.484
C06688=1143.181,-113.372,-43.887,178.624,6.004,149.484
C06689=1143.186,-113.622,-43.878,178.622,6.004,149.485
C06690=1143.192,-113.872,-43.870,178.620,6.004,149.485
C06691=1143.198,-114.121,-43.861,178.618,6.003,149.486
C06692=1143.203,-114.371,-43.852,178.616,6.003,149.486
C06693=1143.208,-114.621,-43.843,178.614,6.002,149.487
C06694=1143.214,-114.870,-43.835,178.612,6.001,149.487
C06695=1143.219,-115.121,-43.827,178.610,6.001,149.488
C06696=1143.224,-115.371,-43.818,178.608,6.001,149.488
C06697=1143.229,-115.620,-43.809,178.606,6.001,149.489
C06698=1143.235,-115.870,-43.800,178.604,6.000,149.489
C06699=1143.240,-116.119,-43.792,178.602,6.000,149.490
C06700=1143.246,-116.370,-43.783,178.600,6.000,149.490
C06701=1143.252,-116.619,-43.775,178.598,6.000,149.491
C06702=1143.257,-116.869,-43.766,178.596,5.999,149.491
C06703=1143.262,-117.119,-43.758,178.594,5.998,149.492
C06704=1143.268,-117.368,-43.749,178.592,5.998,149.492
C06705=1143.273,-117.618,-43.740,178.590,5.998,149.493
C06706=1143.278,-117.868,-43.731,178.588,5.998,149.493
C06707=1143.284,-118.119,-43.723,178.586,5.997,149.494
C06708=1143.290,-118.368,-43.715,178.585,5.997,149.494
C06709=1143.295,-118.618,-43.706,178.582,5.996,149.495
C06710=1143.299,-118.868,-43.698,178.581,5.996,149.495
C06711=1143.305,-119.117,-43.690,178.579,5.995,149.496
C06712=1143.310,-119.367,-43.681,178.577,5.995,149.496
C06713=1143.316,-119.617,-43.672,178.575,5.995,149.497
C06714=1143.322,-119.866,-43.664,178.572,5.994,149.497
C06715=1143.327,-120.116,-43.655,178.571,5.994,149.498
C06716=1143.332,-120.366,-43.646,178.568,5.994,149.498
C06717=1143.338,-120.616,-43.638,178.567,5.994,149.499
C06718=1143.343,-120.866,-43.630,178.565,5.993,149.499
C06719=1143.348,-121.116,-43.622,178.563,5.993,149.500
C06720=1143.354,-121.365,-43.613,178.561,5.992,149.500
C06721=1143.359,-121.615,-43.605,178.559,5.992,149.501
C06722=1143.364,-121.865,-43.596,178.557,5.992,149.501
C06723=1143.370,-122.115,-43.588,178.555,5.992,149.502
C06724=1143.375,-122.364,-43.579,178.553,5.991,149.502
C06725=1143.381,-122.615,-43.571,178.552,5.991,149.503
C06726=1143.386,-122.864,-43.563,178.549,5.990,149.503
C06727=1143.391,-123.114,-43.555,178.548,5.990,149.504
C06728=1143.396,-123.364,-43.546,178.546,5.989,149.504
C06729=1143.402,-123.613,-43.537,178.544,5.990,149.505
C06730=1143.408,-123.864,-43.529,178.542,5.989,149.505
C06731=1143.413,-124.113,-43.520,178.540,5.988,149.506
C06732=1143.418,-124.363,-43.513,178.538,5.988,149.506
C06733=1143.423,-124.613,-43.504,178.536,5.987,149.507
C06734=1143.429,-124.863,-43.496,178.534,5.987,149.507
C06735=1143.435,-125.112,-43.487,178.532,5.987,149.508
C06736=1143.440,-125.363,-43.479,178.530,5.987,149.508
C06737=1143.445,-125.612,-43.471,178.528,5.986,149.509
C06738=1143.451,-125.862,-43.463,178.527,5.986,149.509
C06739=1143.456,-126.111,-43.454,178.524,5.985,149.510
C06740=1143.462,-126.362,-43.446,178.523,5.985,149.510
C06741=1143.467,-126.612,-43.437,178.521,5.985,149.510
C06742=1143.472,-126.861,-43.430,178.519,5.985,149.511
C06743=1143.477,-127.111,-43.421,178.516,5.984,149.512
C06744=1143.484,-127.361,-43.413,178.515,5.984,149.512
C06745=1143.489,-127.611,-43.405,178.513,5.984,149.513
C06746=1143.494,-127.860,-43.397,178.511,5.984,149.513
C06747=1143.499,-128.110,-43.388,178.509,5.983,149.514
C06748=1143.505,-128.360,-43.380,178.507,5.983,149.514
C06749=1143.084,-128.371,-43.423,178.504,5.986,149.516
C06750=1143.079,-128.121,-43.432,178.506,5.986,149.515
C06751=1143.073,-127.872,-43.440,178.508,5.986,149.515
C06752=1143.068,-127.622,-43.449,178.510,5.987,149.514
C06753=1143.062,-127.372,-43.456,178.511,5.987,149.514
C06754=1143.057,-127.122,-43.465,178.514,5.988,149.513
C06755=1143.052,-126.872,-43.473,178.515,5.988,149.513
C06756=1143.046,-126.622,-43.481,178.517,5.989,149.512
C06757=1143.040,-126.372,-43.490,178.519,5.989,149.512
C06758=1143.035,-126.123,-43.498,178.521,5.989,149.511
C06759=1143.030,-125.873,-43.506,178.523,5.989,149.511
C06760=1143.025,-125.623,-43.515,178.525,5.990,149.510
C06761=1143.019,-125.373,-43.523,178.527,5.990,149.510
C06762=1143.013,-125.124,-43.531,178.529,5.991,149.509
C06763=1143.008,-124.874,-43.539,178.530,5.991,149.509
C06764=1143.003,-124.624,-43.548,178.533,5.991,149.508
C06765=1142.998,-124.374,-43.556,178.534,5.991,149.508
C06766=1142.992,-124.125,-43.564,178.536,5.992,149.507
C06767=1142.986,-123.874,-43.572,178.538,5.992,149.507
C06768=1142.981,-123.625,-43.580,178.540,5.993,149.506
C06769=1142.976,-123.375,-43.589,178.542,5.994,149.506
C06770=1142.971,-123.125,-43.597,178.544,5.993,149.505
C06771=1142.965,-122.876,-43.606,178.546,5.994,149.505
C06772=1142.959,-122.625,-43.614,178.548,5.994,149.504
C06773=1142.954,-122.376,-43.623,178.550,5.995,149.504
C06774=1142.949,-122.126,-43.630,178.552,5.995,149.504
C06775=1142.944,-121.876,-43.639,178.554,5.996,149.503
C06776=1142.939,-121.626,-43.648,178.555,5.996,149.503
C06777=1142.932,-121.377,-43.656,178.558,5.996,149.502
C06778=1142.927,-121.127,-43.665,178.559,5.996,149.502
C06779=1142.922,-120.877,-43.674,178.561,5.997,149.501
C06780=1142.916,-120.627,-43.682,178.563,5.997,149.500
C06781=1142.912,-120.378,-43.690,178.566,5.997,149.500
C06782=1142.906,-120.127,-43.698,178.567,5.997,149.499
C06783=1142.900,-119.878,-43.707,178.569,5.998,149.499
C06784=1142.895,-119.628,-43.715,178.572,5.999,149.498
C06785=1142.890,-119.378,-43.724,178.573,5.999,149.498
C06786=1142.884,-119.128,-43.732,178.575,5.999,149.497
C06787=1142.879,-118.879,-43.741,178.577,5.999,149.497
C06788=1142.874,-118.629,-43.750,178.579,6.000,149.496
C06789=1142.868,-118.379,-43.758,178.581,6.000,149.496
C06790=1142.862,-118.129,-43.767,178.583,6.001,149.495
C06791=1142.858,-117.880,-43.775,178.585,6.001,149.495
C06792=1142.852,-117.630,-43.783,178.587,6.002,149.495
C06793=1142.847,-117.380,-43.792,178.588,6.002,149.494
C06794=1142.842,-117.130,-43.801,178.591,6.002,149.494
C06795=1142.836,-116.880,-43.809,178.593,6.003,149.493
C06796=1142.830,-116.631,-43.817,178.594,6.003,149.493
C06797=1142.825,-116.381,-43.826,178.597,6.004,149.492
C06798=1142.820,-116.131,-43.835,178.599,6.003,149.491
C06799=1142.814,-115.882,-43.844,178.601,6.004,149.491
C06800=1142.809,-115.631,-43.852,178.602,6.004,149.490
C06801=1142.804,-115.381,-43.861,178.605,6.005,149.490
C06802=1142.798,-115.132,-43.870,178.606,6.005,149.489
C06803=1142.793,-114.882,-43.878,178.608,6.006,149.489
C06804=1142.787,-114.632,-43.886,178.611,6.006,149.488
C06805=1142.782,-114.382,-43.895,178.612,6.006,149.488
C06806=1142.776,-114.133,-43.904,178.614,6.007,149.487
C06807=1142.771,-113.883,-43.913,178.616,6.007,149.487
C06808=1142.766,-113.633,-43.922,178.618,6.008,149.486
C06809=1142.760,-113.383,-43.930,178.620,6.008,149.486
C06810=1142.755,-113.134,-43.938,178.623,6.008,149.485
C06811=1142.750,-112.884,-43.947,178.624,6.008,149.485
C06812=1142.744,-112.634,-43.956,178.626,6.009,149.484
C06813=1142.739,-112.384,-43.965,178.629,6.009,149.484
C06814=1142.733,-112.135,-43.973,178.630,6.009,149.483
C06815=1142.728,-111.884,-43.982,178.632,6.010,149.483
C06816=1142.723,-111.635,-43.991,178.634,6.010,149.482
C06817=1142.718,-111.385,-43.999,178.636,6.011,149.482
C06818=1142.712,-111.135,-44.008,178.638,6.011,149.481
C06819=1142.707,-110.886,-44.017,178.640,6.012,149.481
C06820=1142.702,-110.636,-44.026,178.642,6.012,149.480
C06821=1142.696,-110.386,-44.035,178.644,6.012,149.480
C06822=1142.690,-110.136,-44.044,178.646,6.013,149.479
C06823=1142.685,-109.886,-44.053,178.648,6.013,149.479
C06824=1142.680,-109.637,-44.062,178.650,6.013,149.478
C06825=1142.674,-109.386,-44.070,178.652,6.014,149.478
C06826=1142.669,-109.136,-44.079,178.654,6.014,149.477
C06827=1142.664,-108.887,-44.088,178.656,6.015,149.477
C06828=1142.659,-108.637,-44.096,178.658,6.015,149.476
C06829=1142.653,-108.388,-44.105,178.660,6.016,149.476
C06830=1142.648,-108.138,-44.114,178.663,6.016,149.475
C06831=1142.642,-107.888,-44.123,178.664,6.016,149.475
C06832=1142.637,-107.638,-44.132,178.666,6.017,149.474
C06833=1142.631,-107.388,-44.141,178.668,6.017,149.474
C06834=1142.626,-107.138,-44.150,178.670,6.017,149.473
C06835=1142.620,-106.889,-44.159,178.672,6.017,149.473
C06836=1142.615,-106.639,-44.168,178.674,6.018,149.472
C06837=1142.610,-106.389,-44.176,178.676,6.019,149.472
C06838=1142.605,-106.139,-44.185,178.678,6.019,149.471
C06839=1142.600,-105.890,-44.194,178.680,6.019,149.471
C06840=1142.594,-105.639,-44.204,178.682,6.019,149.470
C06841=1142.588,-105.390,-44.212,178.684,6.020,149.470
C06842=1142.583,-105.140,-44.221,178.686,6.021,149.469
C06843=1142.578,-104.891,-44.230,178.688,6.021,149.469
C06844=1142.573,-104.641,-44.239,178.690,6.021,149.468
C06845=1142.567,-104.391,-44.248,178.692,6.022,149.468
C06846=1142.562,-104.141,-44.257,178.695,6.022,149.467
C06847=1142.556,-103.891,-44.266,178.697,6.022,149.466
C06848=1142.551,-103.641,-44.275,178.698,6.022,149.466
C06849=1142.546,-103.392,-44.284,178.701,6.023,149.465
C06850=1142.540,-103.120,-44.294,178.703,6.024,149.465
C06851=1142.534,-102.848,-44.304,178.705,6.023,149.464
C06852=1142.529,-102.575,-44.314,178.707,6.024,149.464
C06853=1142.522,-102.303,-44.324,178.709,6.025,149.463
C06854=1142.517,-102.053,-44.333,178.711,6.026,149.463
C06855=1142.512,-101.803,-44.342,178.713,6.025,149.462
C06856=1142.507,-101.554,-44.351,178.716,6.026,149.462
C06857=1142.501,-101.304,-44.360,178.717,6.026,149.461
C06858=1142.495,-101.054,-44.369,178.719,6.027,149.461
C06859=1142.490,-100.804,-44.378,178.722,6.027,149.460
C06860=1142.485,-100.555,-44.387,178.723,6.027,149.460
C06861=1142.480,-100.305,-44.397,178.725,6.028,149.459
C06862=1142.474,-100.055,-44.406,178.728,6.028,149.458
C06863=1142.469,-99.805,-44.415,178.730,6.028,149.458
C06864=1142.464,-99.555,-44.424,178.732,6.029,149.457
C06865=1142.458,-99.305,-44.433,178.734,6.030,149.457
C06866=1142.453,-99.055,-44.442,178.736,6.030,149.456
C06867=1142.448,-98.806,-44.452,178.738,6.031,149.456
C06868=1142.443,-98.556,-44.461,178.740,6.030,149.455
C06869=1142.437,-98.306,-44.470,178.742,6.031,149.455
C06870=1142.432,-98.056,-44.479,178.744,6.032,149.454
C06871=1142.426,-97.808,-44.488,178.746,6.032,149.454
C06872=1142.420,-97.558,-44.498,178.748,6.032,149.453
C06873=1142.415,-97.308,-44.507,178.750,6.033,149.453
C06874=1142.410,-97.058,-44.516,178.752,6.033,149.452
C06875=1142.404,-96.808,-44.525,178.755,6.034,149.452
C06876=1142.399,-96.559,-44.535,178.757,6.034,149.451
C06877=1142.394,-96.309,-44.544,178.758,6.034,149.451
C06878=1142.388,-96.059,-44.553,178.761,6.035,149.450
C06879=1142.383,-95.809,-44.563,178.762,6.035,149.450
C06880=1142.378,-95.559,-44.572,178.765,6.035,149.449
C06881=1142.372,-95.309,-44.581,178.767,6.036,149.449
C06882=1142.367,-95.059,-44.590,178.769,6.036,149.448
C06883=1142.362,-94.810,-44.600,178.771,6.037,149.448
C06884=1142.356,-94.560,-44.609,178.773,6.038,149.447
C06885=1142.351,-94.310,-44.618,178.775,6.038,149.447
C06886=1142.346,-94.061,-44.628,178.777,6.038,149.446
C06887=1142.340,-93.811,-44.637,178.780,6.039,149.445
C06888=1142.335,-93.561,-44.646,178.781,6.039,149.445
C06889=1142.330,-93.311,-44.656,178.783,6.039,149.444
C06890=1142.324,-93.062,-44.665,178.786,6.040,149.444
C06891=1142.319,-92.812,-44.674,178.788,6.040,149.443
C06892=1142.314,-92.562,-44.684,178.790,6.041,149.443
C06893=1142.308,-92.312,-44.693,178.792,6.041,149.442
C06894=1142.303,-92.063,-44.703,178.794,6.041,149.442
C06895=1142.298,-91.813,-44.712,178.796,6.042,149.441
C06896=1142.292,-91.563,-44.722,178.798,6.043,149.441
C06897=1142.287,-91.314,-44.731,178.800,6.042,149.440
C06898=1142.282,-91.064,-44.740,178.802,6.043,149.440
C06899=1142.276,-90.814,-44.751,178.804,6.044,149.439
C06900=1142.271,-90.564,-44.759,178.806,6.044,149.439
C06901=1142.266,-90.313,-44.769,178.808,6.045,149.438
C06902=1142.261,-90.064,-44.779,178.811,6.045,149.437
C06903=1142.255,-89.814,-44.788,178.812,6.045,149.437
C06904=1142.250,-89.565,-44.798,178.815,6.046,149.436
C06905=1142.244,-89.315,-44.807,178.817,6.046,149.436
C06906=1142.239,-89.065,-44.817,178.819,6.047,149.435
C06907=1142.234,-88.816,-44.826,178.821,6.047,149.435
C06908=1142.229,-88.566,-44.836,178.823,6.048,149.434
C06909=1142.223,-88.316,-44.845,178.826,6.048,149.434
C06910=1142.218,-88.067,-44.855,178.827,6.048,149.433
C06911=1142.213,-87.817,-44.864,178.829,6.049,149.433
C06912=1142.207,-87.567,-44.874,178.832,6.049,149.432
C06913=1142.202,-87.317,-44.883,178.834,6.049,149.432
C06914=1142.197,-87.067,-44.894,178.836,6.050,149.431
C06915=1142.192,-86.817,-44.903,178.838,6.051,149.431
C06916=1142.186,-86.568,-44.913,178.840,6.051,149.430
C06917=1142.181,-86.318,-44.922,178.842,6.051,149.429
C06918=1142.175,-86.068,-44.932,178.844,6.052,149.429
C06919=1142.170,-85.819,-44.941,178.846,6.052,149.429
C06920=1142.165,-85.569,-44.951,178.848,6.053,149.428
C06921=1142.159,-85.319,-44.961,178.851,6.053,149.427
C06922=1142.154,-85.070,-44.970,178.853,6.054,149.427
C06923=1142.149,-84.819,-44.981,178.855,6.054,149.426
C06924=1142.144,-84.569,-44.990,178.857,6.055,149.426
C06925=1142.138,-84.320,-45.000,178.859,6.055,149.425
C06926=1142.133,-84.070,-45.009,178.861,6.055,149.425
C06927=1142.127,-83.821,-45.019,178.863,6.056,149.424
C06928=1142.122,-83.571,-45.029,178.866,6.056,149.424
C06929=1142.116,-83.321,-45.038,178.868,6.057,149.423
C06930=1142.111,-83.071,-45.049,178.870,6.057,149.423
C06931=1142.106,-82.821,-45.058,178.872,6.058,149.422
C06932=1142.101,-82.572,-45.068,178.874,6.058,149.422
C06933=1142.096,-82.322,-45.078,178.876,6.058,149.421
C06934=1142.090,-82.072,-45.087,178.878,6.059,149.421
C06935=1142.084,-81.823,-45.097,178.881,6.059,149.420
C06936=1142.080,-81.573,-45.107,178.883,6.060,149.419
C06937=1142.074,-81.322,-45.117,178.884,6.060,149.419
C06938=1142.069,-81.073,-45.127,178.887,6.061,149.418
C06939=1142.064,-80.824,-45.137,178.889,6.061,149.418
C06940=1142.058,-80.574,-45.146,178.891,6.061,149.417
C06941=1142.053,-80.324,-45.156,178.893,6.062,149.417
C06942=1142.048,-80.074,-45.166,178.895,6.063,149.416
C06943=1142.042,-79.825,-45.176,178.898,6.063,149.416
C06944=1142.037,-79.575,-45.185,178.900,6.063,149.415
C06945=1142.032,-79.325,-45.195,178.902,6.064,149.415
C06946=1142.026,-79.076,-45.206,178.904,6.065,149.414
C06947=1142.021,-78.825,-45.215,178.907,6.065,149.413
C06948=1142.016,-78.575,-45.225,178.908,6.065,149.413
C06949=1142.010,-78.326,-45.235,178.910,6.066,149.412
C06950=1142.005,-78.076,-45.246,178.913,6.066,149.412
C06951=1141.999,-77.827,-45.254,178.915,6.067,149.411
C06952=1141.994,-77.576,-45.265,178.917,6.067,149.411
C06953=1141.989,-77.327,-45.275,178.919,6.068,149.410
C06954=1141.984,-77.055,-45.286,178.921,6.068,149.410
C06955=1141.977,-76.784,-45.297,178.924,6.069,149.409
C06956=1141.972,-76.513,-45.308,178.926,6.069,149.409
C06957=1141.967,-76.241,-45.319,178.929,6.070,149.408
C06958=1141.961,-75.992,-45.329,178.930,6.070,149.407
C06959=1141.955,-75.742,-45.338,178.933,6.071,149.407
C06960=1141.949,-75.492,-45.348,178.935,6.071,149.406
C06961=1141.944,-75.242,-45.359,178.937,6.072,149.406
C06962=1141.940,-74.993,-45.369,178.939,6.072,149.405
C06963=1141.934,-74.743,-45.379,178.941,6.072,149.405
C06964=1141.928,-74.494,-45.389,178.944,6.073,149.404
C06965=1141.923,-74.243,-45.399,178.946,6.074,149.404
C06966=1141.918,-73.993,-45.409,178.948,6.074,149.403
C06967=1141.913,-73.744,-45.419,178.950,6.074,149.403
C06968=1141.907,-73.494,-45.429,178.953,6.075,149.402
C06969=1141.902,-73.244,-45.440,178.955,6.076,149.401
C06970=1141.896,-72.995,-45.450,178.956,6.075,149.401
C06971=1141.892,-72.745,-45.459,178.958,6.076,149.400
C06972=1141.887,-72.495,-45.470,178.961,6.077,149.400
C06973=1141.881,-72.246,-45.480,178.963,6.077,149.399
C06974=1141.875,-71.996,-45.490,178.966,6.078,149.399
C06975=1141.870,-71.746,-45.501,178.967,6.078,149.398
C06976=1141.865,-71.496,-45.510,178.970,6.079,149.398
C06977=1141.860,-71.246,-45.520,178.972,6.079,149.397
C06978=1141.854,-70.997,-45.530,178.974,6.080,149.397
C06979=1141.849,-70.747,-45.541,178.976,6.080,149.396
C06980=1141.843,-70.497,-45.551,178.978,6.080,149.395
C06981=1141.838,-70.247,-45.561,178.981,6.081,149.395
C06982=1141.833,-69.997,-45.572,178.983,6.082,149.394
C06983=1141.828,-69.748,-45.581,178.986,6.082,149.394
C06984=1141.822,-69.498,-45.592,178.987,6.082,149.393
C06985=1141.817,-69.248,-45.602,178.989,6.083,149.393
C06986=1141.812,-68.999,-45.612,178.992,6.084,149.392
C06987=1141.806,-68.749,-45.623,178.994,6.084,149.392
C06988=1141.801,-68.499,-45.633,178.996,6.085,149.391
C06989=1141.796,-68.249,-45.643,178.998,6.085,149.391
C06990=1141.790,-68.000,-45.654,179.001,6.085,149.390
C06991=1141.785,-67.750,-45.665,179.003,6.086,149.389
C06992=1141.780,-67.501,-45.675,179.005,6.087,149.389
C06993=1141.775,-67.251,-45.685,179.007,6.087,149.389
C06994=1141.770,-67.001,-45.695,179.009,6.087,149.388
C06995=1141.764,-66.752,-45.706,179.011,6.088,149.387
C06996=1141.759,-66.501,-45.716,179.014,6.089,149.387
C06997=1141.754,-66.252,-45.726,179.016,6.089,149.386
C06998=1141.748,-66.002,-45.736,179.018,6.089,149.386
C06999=1141.743,-65.752,-45.747,179.020,6.090,149.385
C07000=1141.737,-65.502,-45.757,179.022,6.091,149.385
C07001=1141.733,-65.253,-45.769,179.025,6.091,149.384
C07002=1141.727,-65.003,-45.779,179.027,6.092,149.384
C07003=1141.722,-64.754,-45.789,179.029,6.093,149.383
C07004=1141.717,-64.504,-45.800,179.031,6.092,149.382
C07005=1141.711,-64.254,-45.810,179.034,6.093,149.382
C07006=1141.706,-64.004,-45.820,179.036,6.094,149.381
C07007=1141.700,-63.754,-45.831,179.038,6.094,149.381
C07008=1141.695,-63.505,-45.841,179.041,6.095,149.380
C07009=1141.690,-63.255,-45.852,179.042,6.095,149.380
C07010=1141.684,-63.005,-45.862,179.044,6.096,149.379
C07011=1141.679,-62.755,-45.873,179.047,6.096,149.379
C07012=1141.674,-62.506,-45.883,179.049,6.097,149.378
C07013=1141.669,-62.256,-45.894,179.052,6.098,149.378
C07014=1141.664,-62.007,-45.905,179.054,6.098,149.377
C07015=1141.658,-61.757,-45.915,179.056,6.098,149.376
C07016=1141.653,-61.507,-45.925,179.058,6.099,149.376
C07017=1141.648,-61.258,-45.936,179.060,6.099,149.375
C07018=1141.643,-61.008,-45.947,179.063,6.100,149.375
C07019=1141.637,-60.758,-45.957,179.065,6.101,149.374
C07020=1141.632,-60.508,-45.968,179.067,6.101,149.374
C07021=1141.627,-60.259,-45.979,179.069,6.101,149.373
C07022=1141.622,-60.009,-45.989,179.071,6.102,149.373
C07023=1141.616,-59.759,-45.999,179.074,6.103,149.372
C07024=1141.611,-59.509,-46.011,179.076,6.103,149.371
C07025=1141.606,-59.260,-46.021,179.079,6.104,149.371
C07026=1141.601,-59.010,-46.031,179.081,6.104,149.370
C07027=1141.596,-58.761,-46.042,179.082,6.104,149.370
C07028=1141.591,-58.510,-46.053,179.085,6.105,149.369
C07029=1141.584,-58.261,-46.064,179.087,6.106,149.369
C07030=1141.580,-58.011,-46.075,179.089,6.106,149.368
C07031=1141.574,-57.761,-46.085,179.092,6.107,149.368
C07032=1141.569,-57.511,-46.096,179.094,6.108,149.367
C07033=1141.564,-57.262,-46.107,179.096,6.108,149.367
C07034=1141.559,-57.012,-46.117,179.098,6.108,149.366
C07035=1141.553,-56.763,-46.127,179.101,6.109,149.365
C07036=1141.548,-56.513,-46.139,179.103,6.109,149.365
C07037=1141.543,-56.263,-46.149,179.106,6.110,149.364
C07038=1141.537,-56.013,-46.161,179.108,6.111,149.364
C07039=1141.532,-55.764,-46.171,179.110,6.111,149.363
C07040=1141.527,-55.514,-46.182,179.112,6.111,149.363
C07041=1141.521,-55.265,-46.193,179.114,6.112,149.362
C07042=1141.516,-55.014,-46.203,179.116,6.113,149.362
C07043=1141.512,-54.765,-46.214,179.119,6.113,149.361
C07044=1141.505,-54.515,-46.225,179.121,6.114,149.360
C07045=1141.501,-54.265,-46.237,179.123,6.114,149.360
C07046=1141.495,-54.016,-46.247,179.126,6.115,149.359
C07047=1141.490,-53.766,-46.258,179.128,6.116,149.359
C07048=1141.485,-53.517,-46.268,179.130,6.116,149.358
C07049=1141.479,-53.266,-46.279,179.132,6.116,149.358
C07050=1141.474,-53.016,-46.291,179.135,6.117,149.357
C07051=1141.469,-52.767,-46.301,179.137,6.118,149.357
C07052=1141.464,-52.517,-46.312,179.139,6.118,149.356
C07053=1141.459,-52.268,-46.323,179.142,6.119,149.355
C07054=1141.453,-52.018,-46.334,179.144,6.119,149.355
C07055=1141.448,-51.769,-46.345,179.146,6.120,149.354
C07056=1141.443,-51.519,-46.356,179.148,6.120,149.354
C07057=1141.438,-51.269,-46.367,179.150,6.121,149.353
C07058=1141.432,-50.999,-46.379,179.153,6.121,149.353
C07059=1141.426,-50.727,-46.390,179.155,6.122,149.352
C07060=1141.420,-50.456,-46.403,179.159,6.123,149.351
C07061=1141.414,-50.186,-46.415,179.161,6.124,149.351
C07062=1141.409,-49.936,-46.426,179.162,6.124,149.350
C07063=1141.404,-49.687,-46.436,179.165,6.124,149.350
C07064=1141.399,-49.437,-46.447,179.167,6.125,149.349
C07065=1141.394,-49.187,-46.459,179.169,6.126,149.349
C07066=1141.388,-48.938,-46.470,179.172,6.126,149.348
C07067=1141.383,-48.688,-46.481,179.174,6.127,149.348
C07068=1141.378,-48.437,-46.492,179.176,6.128,149.347
C07069=1141.372,-48.188,-46.503,179.179,6.128,149.346
C07070=1141.368,-47.939,-46.514,179.181,6.129,149.346
C07071=1141.361,-47.689,-46.525,179.183,6.130,149.345
C07072=1141.357,-47.439,-46.536,179.185,6.129,149.345
C07073=1141.352,-47.190,-46.548,179.188,6.130,149.344
C07074=1141.346,-46.940,-46.558,179.190,6.131,149.344
C07075=1141.341,-46.690,-46.570,179.193,6.131,149.343
C07076=1141.336,-46.441,-46.581,179.195,6.132,149.343
C07077=1141.330,-46.191,-46.592,179.197,6.133,149.342
C07078=1141.325,-45.941,-46.603,179.200,6.133,149.341
C07079=1141.321,-45.692,-46.614,179.202,6.134,149.341
C07080=1141.315,-45.442,-46.626,179.204,6.135,149.341
C07081=1141.310,-45.192,-46.636,179.207,6.135,149.340
C07082=1141.304,-44.942,-46.648,179.209,6.136,149.339
C07083=1141.299,-44.692,-46.660,179.211,6.137,149.339
C07084=1141.294,-44.444,-46.671,179.213,6.136,149.338
C07085=1141.288,-44.193,-46.682,179.215,6.137,149.338
C07086=1141.284,-43.943,-46.693,179.218,6.137,149.337
C07087=1141.278,-43.694,-46.705,179.220,6.138,149.336
C07088=1141.273,-43.445,-46.716,179.222,6.139,149.336
C07089=1141.267,-43.194,-46.727,179.225,6.139,149.335
C07090=1141.263,-42.944,-46.738,179.227,6.140,149.335
C07091=1141.257,-42.695,-46.749,179.229,6.141,149.334
C07092=1141.252,-42.445,-46.761,179.232,6.141,149.334
C07093=1141.247,-42.196,-46.772,179.234,6.142,149.333
C07094=1141.241,-41.947,-46.784,179.236,6.143,149.333
C07095=1141.236,-41.696,-46.794,179.239,6.143,149.332
C07096=1141.231,-41.446,-46.806,179.241,6.144,149.332
C07097=1141.226,-41.197,-46.818,179.243,6.145,149.331
C07098=1141.220,-40.948,-46.829,179.246,6.145,149.330
C07099=1141.215,-40.698,-46.840,179.248,6.146,149.330
C07100=1141.210,-40.448,-46.852,179.250,6.146,149.329
C07101=1141.205,-40.198,-46.864,179.252,6.146,149.329
C07102=1141.199,-39.949,-46.874,179.255,6.147,149.328
C07103=1141.194,-39.699,-46.886,179.257,6.148,149.328
C07104=1141.189,-39.449,-46.898,179.260,6.148,149.327
C07105=1141.184,-39.199,-46.909,179.262,6.149,149.327
C07106=1141.179,-38.949,-46.921,179.264,6.150,149.326
C07107=1141.173,-38.701,-46.932,179.267,6.150,149.325
C07108=1141.168,-38.451,-46.944,179.269,6.151,149.325
C07109=1141.163,-38.201,-46.955,179.271,6.152,149.324
C07110=1141.158,-37.951,-46.967,179.274,6.152,149.324
C07111=1141.152,-37.702,-46.978,179.276,6.153,149.323
C07112=1141.147,-37.452,-46.990,179.278,6.153,149.323
C07113=1141.142,-37.202,-47.001,179.281,6.154,149.322
C07114=1141.137,-36.953,-47.013,179.283,6.155,149.322
C07115=1141.131,-36.703,-47.025,179.286,6.155,149.321
C07116=1141.126,-36.454,-47.036,179.288,6.156,149.320
C07117=1141.121,-36.204,-47.047,179.290,6.157,149.320
C07118=1141.116,-35.954,-47.059,179.293,6.157,149.319
C07119=1141.111,-35.704,-47.071,179.295,6.158,149.319
C07120=1141.105,-35.454,-47.082,179.297,6.159,149.318
C07121=1141.100,-35.205,-47.094,179.300,6.159,149.318
C07122=1141.094,-34.955,-47.105,179.302,6.160,149.317
C07123=1141.089,-34.705,-47.117,179.304,6.161,149.316
C07124=1141.084,-34.456,-47.128,179.307,6.161,149.316
C07125=1141.079,-34.206,-47.140,179.309,6.162,149.315
C07126=1141.074,-33.956,-47.152,179.311,6.163,149.315
C07127=1141.069,-33.706,-47.164,179.314,6.163,149.314
C07128=1141.063,-33.456,-47.175,179.316,6.164,149.314
C07129=1141.058,-33.208,-47.186,179.319,6.165,149.313
C07130=1141.053,-32.958,-47.199,179.321,6.165,149.313
C07131=1141.048,-32.708,-47.211,179.323,6.166,149.312
C07132=1141.043,-32.459,-47.222,179.326,6.166,149.311
C07133=1141.037,-32.209,-47.234,179.328,6.167,149.311
C07134=1141.032,-31.959,-47.246,179.330,6.168,149.310
C07135=1141.027,-31.709,-47.257,179.333,6.168,149.310
C07136=1141.022,-31.459,-47.269,179.335,6.169,149.309
C07137=1141.016,-31.211,-47.281,179.337,6.170,149.309
C07138=1141.011,-30.961,-47.293,179.340,6.170,149.308
C07139=1141.006,-30.711,-47.304,179.342,6.171,149.308
C07140=1141.001,-30.461,-47.316,179.344,6.172,149.307
C07141=1140.995,-30.211,-47.328,179.347,6.172,149.307
C07142=1140.991,-29.962,-47.340,179.349,6.173,149.306
C07143=1140.985,-29.712,-47.352,179.351,6.174,149.305
C07144=1140.980,-29.462,-47.364,179.354,6.174,149.305
C07145=1140.974,-29.212,-47.376,179.356,6.175,149.304
C07146=1140.970,-28.963,-47.387,179.359,6.176,149.304
C07147=1140.965,-28.713,-47.400,179.361,6.176,149.303
C07148=1140.959,-28.463,-47.412,179.363,6.177,149.303
C07149=1140.954,-28.213,-47.424,179.366,6.178,149.302
C07150=1140.949,-27.964,-47.435,179.368,6.178,149.302
C07151=1140.944,-27.715,-47.447,179.370,6.179,149.301
C07152=1140.938,-27.465,-47.459,179.373,6.180,149.300
C07153=1140.933,-27.215,-47.471,179.375,6.180,149.300
C07154=1140.928,-26.966,-47.483,179.377,6.181,149.299
C07155=1140.923,-26.716,-47.495,179.380,6.182,149.299
C07156=1140.917,-26.467,-47.507,179.382,6.182,149.298
C07157=1140.912,-26.217,-47.519,179.384,6.183,149.298
C07158=1140.907,-25.967,-47.531,179.387,6.184,149.297
C07159=1140.902,-25.718,-47.542,179.389,6.184,149.296
C07160=1140.897,-25.468,-47.555,179.391,6.185,149.296
C07161=1140.891,-25.218,-47.567,179.394,6.185,149.295
C07162=1140.886,-24.948,-47.580,179.396,6.186,149.295
C07163=1140.881,-24.678,-47.593,179.400,6.187,149.294
C07164=1140.874,-24.408,-47.606,179.402,6.188,149.294
C07165=1140.869,-24.138,-47.620,179.404,6.188,149.293
C07166=1140.864,-23.888,-47.632,179.407,6.189,149.292
C07167=1140.858,-23.638,-47.643,179.409,6.190,149.292
C07168=1140.853,-23.389,-47.656,179.411,6.190,149.291
C07169=1140.849,-23.139,-47.667,179.414,6.191,149.291
C07170=1140.843,-22.890,-47.680,179.416,6.192,149.290
C07171=1140.838,-22.640,-47.692,179.418,6.192,149.290
C07172=1140.833,-22.391,-47.704,179.421,6.193,149.289
C07173=1140.827,-22.141,-47.716,179.423,6.194,149.289
C07174=1140.822,-21.891,-47.729,179.426,6.195,149.288
C07175=1140.817,-21.641,-47.741,179.429,6.196,149.287
C07176=1140.811,-21.391,-47.753,179.431,6.196,149.287
C07177=1140.806,-21.142,-47.765,179.433,6.197,149.286
C07178=1140.801,-20.892,-47.777,179.436,6.198,149.286
C07179=1140.796,-20.643,-47.790,179.438,6.198,149.285
C07180=1140.790,-20.393,-47.802,179.440,6.199,149.285
C07181=1140.785,-20.144,-47.814,179.443,6.200,149.284
C07182=1140.781,-19.895,-47.826,179.445,6.200,149.284
C07183=1140.775,-19.645,-47.838,179.448,6.201,149.283
C07184=1140.771,-19.395,-47.851,179.450,6.202,149.282
C07185=1140.765,-19.145,-47.863,179.452,6.202,149.282
C07186=1140.760,-18.895,-47.876,179.455,6.203,149.281
C07187=1140.755,-18.645,-47.888,179.457,6.204,149.281
C07188=1140.750,-18.396,-47.900,179.460,6.205,149.280
C07189=1140.745,-18.147,-47.913,179.462,6.206,149.280
C07190=1140.739,-17.897,-47.925,179.465,6.206,149.279
C07191=1140.734,-17.648,-47.937,179.467,6.207,149.278
C07192=1140.729,-17.398,-47.949,179.469,6.208,149.278
C07193=1140.724,-17.148,-47.962,179.472,6.208,149.278
C07194=1140.719,-16.898,-47.975,179.474,6.209,149.277
C07195=1140.713,-16.648,-47.987,179.476,6.210,149.276
C07196=1140.708,-16.399,-48.000,179.479,6.210,149.276
C07197=1140.703,-16.149,-48.012,179.481,6.211,149.275
C07198=1140.697,-15.899,-48.024,179.483,6.212,149.275
C07199=1140.692,-15.650,-48.037,179.487,6.213,149.274
C07200=1140.687,-15.401,-48.049,179.489,6.214,149.274
C07201=1140.682,-15.150,-48.062,179.491,6.214,149.273
C07202=1140.677,-14.901,-48.074,179.494,6.215,149.272
C07203=1140.672,-14.652,-48.087,179.496,6.216,149.272
C07204=1140.666,-14.402,-48.099,179.499,6.216,149.271
C07205=1140.661,-14.152,-48.111,179.501,6.217,149.271
C07206=1140.656,-13.903,-48.124,179.503,6.218,149.270
C07207=1140.651,-13.654,-48.137,179.506,6.218,149.270
C07208=1140.646,-13.403,-48.149,179.508,6.219,149.269
C07209=1140.640,-13.153,-48.162,179.511,6.220,149.268
C07210=1140.635,-12.904,-48.175,179.513,6.221,149.268
C07211=1140.630,-12.655,-48.187,179.515,6.222,149.268
C07212=1140.625,-12.405,-48.199,179.518,6.222,149.267
C07213=1140.620,-12.155,-48.212,179.520,6.223,149.266
C07214=1140.615,-11.906,-48.225,179.522,6.224,149.266
C07215=1140.610,-11.656,-48.237,179.525,6.224,149.265
C07216=1140.604,-11.407,-48.250,179.527,6.225,149.265
C07217=1140.599,-11.157,-48.262,179.530,6.226,149.264
C07218=1140.594,-10.907,-48.275,179.533,6.227,149.264
C07219=1140.589,-10.657,-48.288,179.535,6.228,149.263
C07220=1140.584,-10.408,-48.301,179.537,6.228,149.262
C07221=1140.579,-10.159,-48.313,179.540,6.229,149.262
C07222=1140.573,-9.908,-48.327,179.542,6.229,149.261
C07223=1140.568,-9.659,-48.339,179.544,6.230,149.261
C07224=1140.563,-9.409,-48.351,179.547,6.232,149.260
C07225=1140.558,-9.160,-48.364,179.550,6.232,149.260
C07226=1140.553,-8.910,-48.377,179.552,6.233,149.259
C07227=1140.547,-8.660,-48.390,179.554,6.234,149.259
C07228=1140.542,-8.411,-48.403,179.557,6.234,149.258
C07229=1140.537,-8.161,-48.415,179.559,6.235,149.258
C07230=1140.533,-7.911,-48.428,179.562,6.235,149.257
C07231=1140.528,-7.662,-48.441,179.565,6.237,149.256
C07232=1140.522,-7.413,-48.454,179.567,6.238,149.256
C07233=1140.517,-7.163,-48.466,179.569,6.238,149.255
C07234=1140.512,-6.913,-48.479,179.572,6.239,149.255
C07235=1140.506,-6.664,-48.493,179.574,6.239,149.254
C07236=1140.501,-6.414,-48.505,179.576,6.240,149.254
C07237=1140.496,-6.164,-48.518,179.579,6.241,149.253
C07238=1140.491,-5.915,-48.531,179.582,6.242,149.252
C07239=1140.486,-5.665,-48.544,179.584,6.243,149.252
C07240=1140.480,-5.416,-48.557,179.587,6.243,149.251
C07241=1140.476,-5.166,-48.570,179.589,6.244,149.251
C07242=1140.470,-4.916,-48.583,179.591,6.245,149.250
C07243=1140.465,-4.667,-48.595,179.594,6.245,149.250
C07244=1140.460,-4.417,-48.608,179.596,6.247,149.249
C07245=1140.454,-4.167,-48.622,179.599,6.248,149.249
C07246=1140.449,-3.918,-48.634,179.601,6.248,149.248
C07247=1140.445,-3.668,-48.647,179.603,6.249,149.248
C07248=1140.439,-3.418,-48.660,179.606,6.250,149.247
C07249=1140.434,-3.169,-48.673,179.609,6.251,149.246
C07250=1140.429,-2.919,-48.686,179.611,6.252,149.246
C07251=1140.423,-2.669,-48.699,179.614,6.252,149.245
C07252=1140.419,-2.421,-48.712,179.616,6.253,149.245
C07253=1140.414,-2.171,-48.725,179.619,6.254,149.244
C07254=1140.408,-1.921,-48.739,179.621,6.254,149.244
C07255=1140.404,-1.671,-48.752,179.624,6.256,149.243
C07256=1140.398,-1.421,-48.765,179.626,6.256,149.242
C07257=1140.393,-1.172,-48.777,179.628,6.257,149.242
C07258=1140.388,-0.922,-48.790,179.631,6.258,149.242
C07259=1140.383,-0.673,-48.804,179.633,6.258,149.241
C07260=1140.378,-0.424,-48.817,179.636,6.260,149.240
C07261=1140.372,-0.173,-48.830,179.639,6.261,149.240
C07262=1140.367,0.076,-48.843,179.641,6.261,149.239
C07263=1140.362,0.326,-48.857,179.643,6.262,149.239
C07264=1140.357,0.575,-48.870,179.646,6.263,149.238
C07265=1140.351,0.825,-48.883,179.648,6.264,149.238
C07266=1140.346,1.094,-48.897,179.651,6.265,149.237
C07267=1140.341,1.364,-48.912,179.653,6.265,149.236
C07268=1140.334,1.633,-48.926,179.657,6.267,149.236
C07269=1140.330,1.902,-48.940,179.659,6.267,149.235
C07270=1140.325,2.152,-48.954,179.661,6.268,149.235
C07271=1140.319,2.402,-48.966,179.664,6.269,149.234
C07272=1140.314,2.651,-48.979,179.667,6.270,149.233
C07273=1140.309,2.901,-48.993,179.669,6.271,149.233
C07274=1140.303,3.150,-49.006,179.671,6.271,149.233
C07275=1140.299,3.400,-49.019,179.674,6.272,149.232
C07276=1140.293,3.649,-49.033,179.677,6.274,149.231
C07277=1140.289,3.899,-49.046,179.679,6.274,149.231
C07278=1140.283,4.149,-49.059,179.681,6.275,149.230
C07279=1140.279,4.399,-49.073,179.684,6.276,149.230
C07280=1140.273,4.648,-49.086,179.687,6.277,149.229
C07281=1140.268,4.898,-49.099,179.689,6.278,149.229
C07282=1140.263,5.147,-49.113,179.692,6.278,149.228
C07283=1140.258,5.398,-49.127,179.694,6.279,149.227
C07284=1140.253,5.646,-49.140,179.697,6.280,149.227
C07285=1140.247,5.897,-49.153,179.699,6.281,149.226
C07286=1140.242,6.146,-49.166,179.701,6.282,149.226
C07287=1140.237,6.396,-49.180,179.704,6.283,149.225
C07288=1140.232,6.645,-49.193,179.707,6.284,149.225
C07289=1140.227,6.895,-49.207,179.709,6.285,149.224
C07290=1140.221,7.144,-49.220,179.712,6.285,149.224
C07291=1140.217,7.394,-49.234,179.714,6.286,149.223
C07292=1140.211,7.643,-49.247,179.717,6.287,149.223
C07293=1140.207,7.893,-49.261,179.719,6.288,149.222
C07294=1140.201,8.142,-49.274,179.721,6.289,149.221
